LIN {X 0,Y 233.584,Z 324.878,A -85,B 0,C 180,E1 -20817.651,E2 -20817.651} C_VEL
LIN {X 0,Y 230.113,Z 315.653,A -85,B 0,C 180,E1 -20819.516,E2 -20819.516} C_VEL
LIN {X 0,Y 226.325,Z 305.069,A -85,B 0,C 180,E1 -20821.384,E2 -20821.384} C_VEL
LIN {X 0,Y 221.321,Z 294.088,A -85,B 0,C 180,E1 -20823.248,E2 -20823.248} C_VEL
LIN {X 0,Y 216.634,Z 285.381,A -85,B 0,C 180,E1 -20824.719,E2 -20824.719} C_VEL
LIN {X 0,Y 215.299,Z 283.034,A -85,B 0,C 180,E1 -20825.102,E2 -20825.102} C_VEL
LIN {X 0,Y 213.881,Z 280.332,A -85,B 0,C 180,E1 -20825.505,E2 -20825.505} C_VEL
LIN {X 0,Y 213.692,Z 279.368,A -85,B 0,C 180,E1 -20825.598,E2 -20825.598} C_VEL
LIN {X 0,Y 213.741,Z 279.36,A -85,B 0,C 180,E1 -20828.662,E2 -20828.662} C_VEL
LIN {X 0,Y 213.757,Z 279.358,A -85,B 0,C 180,E1 -20831.114,E2 -20831.114} C_VEL
LIN {X 0,Y 213.799,Z 279.355,A -85,B 0,C 180,E1 -20833.702,E2 -20833.702} C_VEL
LIN {X 0,Y 213.776,Z 279.356,A -85,B 0,C 180,E1 -20836.358,E2 -20836.358} C_VEL
LIN {X 0,Y 213.763,Z 279.358,A -85,B 0,C 180,E1 -20839.128,E2 -20839.128} C_VEL
LIN {X 0,Y 213.723,Z 279.362,A -85,B 0,C 180,E1 -20843.724,E2 -20843.724} C_VEL
LIN {X 0,Y 213.769,Z 279.357,A -85,B 0,C 180,E1 -20848.735,E2 -20848.735} C_VEL
LIN {X 0,Y 213.802,Z 279.353,A -85,B 0,C 180,E1 -20852.614,E2 -20852.614} C_VEL
LIN {X 0,Y 213.797,Z 279.354,A -85,B 0,C 180,E1 -20856.985,E2 -20856.985} C_VEL
LIN {X 0,Y 213.876,Z 279.345,A -85,B 0,C 180,E1 -20862.811,E2 -20862.811} C_VEL
LIN {X 0,Y 213.921,Z 279.337,A -85,B 0,C 180,E1 -20866.717,E2 -20866.717} C_VEL
LIN {X 0,Y 214.127,Z 279.307,A -85,B 0,C 180,E1 -20870.566,E2 -20870.566} C_VEL
LIN {X 0,Y 214.076,Z 279.315,A -85,B 0,C 180,E1 -20874.359,E2 -20874.359} C_VEL
LIN {X 0,Y 214.402,Z 279.25,A -85,B 0,C 180,E1 -20878.133,E2 -20878.133} C_VEL
LIN {X 0,Y 214.507,Z 279.25,A -85,B 0,C 180,E1 -20880.011,E2 -20880.011} C_VEL
LIN {X 0,Y 214.401,Z 279.275,A -85,B 0,C 180,E1 -20881.889,E2 -20881.889} C_VEL
LIN {X 0,Y 214.183,Z 279.306,A -85,B 0,C 180,E1 -20887.553,E2 -20887.553} C_VEL
LIN {X 0,Y 213.985,Z 279.33,A -85,B 0,C 180,E1 -20891.376,E2 -20891.376} C_VEL
LIN {X 0,Y 213.876,Z 279.344,A -85,B 0,C 180,E1 -20895.251,E2 -20895.251} C_VEL
LIN {X 0,Y 213.798,Z 279.354,A -85,B 0,C 180,E1 -20899.202,E2 -20899.202} C_VEL
LIN {X 0,Y 213.774,Z 279.359,A -85,B 0,C 180,E1 -20903.246,E2 -20903.246} C_VEL
LIN {X 0,Y 213.84,Z 279.719,A -85,B 0,C 180,E1 -20907.405,E2 -20907.405} C_VEL
LIN {X 0,Y 214.016,Z 281.418,A -85,B 0,C 180,E1 -20911.707,E2 -20911.707} C_VEL
LIN {X 0,Y 214.301,Z 283.414,A -85,B 0,C 180,E1 -20916.19,E2 -20916.19} C_VEL
LIN {X 0,Y 214.677,Z 285.89,A -85,B 0,C 180,E1 -20921.153,E2 -20921.153} C_VEL
LIN {X 0,Y 214.856,Z 287.42,A -85,B 0,C 180,E1 -20923.977,E2 -20923.977} C_VEL
LIN {X 0,Y 214.874,Z 288.962,A -85,B 0,C 180,E1 -20926.619,E2 -20926.619} C_VEL
LIN {X 0,Y 214.706,Z 290.501,A -85,B 0,C 180,E1 -20929.107,E2 -20929.107} C_VEL
LIN {X 0,Y 214.243,Z 292.34,A -85,B 0,C 180,E1 -20931.946,E2 -20931.946} C_VEL
LIN {X 0,Y 213.723,Z 294.297,A -85,B 0,C 180,E1 -20934.668,E2 -20934.668} C_VEL
LIN {X 0,Y 214.726,Z 297.663,A -85,B 0,C 180,E1 -20935.037,E2 -20935.037} C_VEL
LIN {X 0,Y 218.182,Z 307.912,A -85,B 0,C 180,E1 -20936.445,E2 -20936.445} C_VEL
LIN {X 0,Y 221.383,Z 321.092,A -85,B 0,C 180,E1 -20938.39,E2 -20938.39} C_VEL
LIN {X 0,Y 222.985,Z 331.539,A -85,B 0,C 180,E1 -20940.079,E2 -20940.079} C_VEL
LIN {X 0,Y 223.807,Z 339.866,A -85,B 0,C 180,E1 -20941.568,E2 -20941.568} C_VEL
LIN {X 0,Y 223.951,Z 349.305,A -85,B 0,C 180,E1 -20943.44,E2 -20943.44} C_VEL
LIN {X 0,Y 223.681,Z 353.86,A -85,B 0,C 180,E1 -20944.405,E2 -20944.405} C_VEL
LIN {X 0,Y 220.756,Z 364.316,A -85,B 0,C 180,E1 -20946.817,E2 -20946.817} C_VEL
LIN {X 0,Y 218.8,Z 371.499,A -85,B 0,C 180,E1 -20948.896,E2 -20948.896} C_VEL
LIN {X 0,Y 216.843,Z 377.815,A -85,B 0,C 180,E1 -20951.089,E2 -20951.089} C_VEL
LIN {X 0,Y 215.402,Z 382.705,A -85,B 0,C 180,E1 -20953.12,E2 -20953.12} C_VEL
LIN {X 0,Y 213.879,Z 385.575,A -85,B 0,C 180,E1 -20954.456,E2 -20954.456} C_VEL
LIN {X 0,Y 209.871,Z 389.592,A -85,B 0,C 180,E1 -20956.645,E2 -20956.645} C_VEL
LIN {X 0,Y 206.107,Z 393.022,A -85,B 0,C 180,E1 -20958.99,E2 -20958.99} C_VEL
LIN {X 0,Y 204.997,Z 394.677,A -85,B 0,C 180,E1 -20960.54,E2 -20960.54} C_VEL
LIN {X 0,Y 204.442,Z 397.502,A -85,B 0,C 180,E1 -20964.081,E2 -20964.081} C_VEL
LIN {X 0,Y 204.364,Z 398.567,A -85,B 0,C 180,E1 -20966.056,E2 -20966.056} C_VEL
LIN {X 0,Y 204.351,Z 399.161,A -85,B 0,C 180,E1 -20968.029,E2 -20968.029} C_VEL
LIN {X 0,Y 204.44,Z 399.319,A -85,B 0,C 180,E1 -20970,E2 -20970} C_VEL
LIN {X 0,Y 204.351,Z 399.161,A -85,B 0,C 180,E1 -20971.971,E2 -20971.971} C_VEL
LIN {X 0,Y 204.374,Z 398.506,A -85,B 0,C 180,E1 -20974.143,E2 -20974.143} C_VEL
LIN {X 0,Y 204.692,Z 396.109,A -85,B 0,C 180,E1 -20977.894,E2 -20977.894} C_VEL
LIN {X 0,Y 205.364,Z 393.153,A -85,B 0,C 180,E1 -20980.849,E2 -20980.849} C_VEL
LIN {X 0,Y 206.41,Z 389.156,A -85,B 0,C 180,E1 -20983.788,E2 -20983.788} C_VEL
LIN {X 0,Y 208.054,Z 384.024,A -85,B 0,C 180,E1 -20986.686,E2 -20986.686} C_VEL
LIN {X 0,Y 209.72,Z 378.758,A -85,B 0,C 180,E1 -20989.07,E2 -20989.07} C_VEL
LIN {X 0,Y 211.801,Z 372.441,A -85,B 0,C 180,E1 -20991.407,E2 -20991.407} C_VEL
LIN {X 0,Y 213.504,Z 366.484,A -85,B 0,C 180,E1 -20993.266,E2 -20993.266} C_VEL
LIN {X 0,Y 215.522,Z 359.556,A -85,B 0,C 180,E1 -20995.082,E2 -20995.082} C_VEL
LIN {X 0,Y 217.202,Z 353.645,A -85,B 0,C 180,E1 -20996.417,E2 -20996.417} C_VEL
LIN {X 0,Y 217.35,Z 343.883,A -85,B 0,C 180,E1 -20998.535,E2 -20998.535} C_VEL
LIN {X 0,Y 216.713,Z 334.568,A -85,B 0,C 180,E1 -21000.347,E2 -21000.347} C_VEL
LIN {X 0,Y 215.482,Z 325.215,A -85,B 0,C 180,E1 -21001.991,E2 -21001.991} C_VEL
LIN {X 0,Y 213.725,Z 316.4,A -85,B 0,C 180,E1 -21003.43,E2 -21003.43} C_VEL
LIN {X 0,Y 210.705,Z 305.251,A -85,B 0,C 180,E1 -21005.113,E2 -21005.113} C_VEL
LIN {X 0,Y 207.594,Z 296.756,A -85,B 0,C 180,E1 -21006.388,E2 -21006.388} C_VEL
LIN {X 0,Y 206.912,Z 293.968,A -85,B 0,C 180,E1 -21006.722,E2 -21006.722} C_VEL
LIN {X 0,Y 207.477,Z 291.775,A -85,B 0,C 180,E1 -21010.06,E2 -21010.06} C_VEL
LIN {X 0,Y 207.716,Z 290.247,A -85,B 0,C 180,E1 -21012.585,E2 -21012.585} C_VEL
LIN {X 0,Y 207.776,Z 288.728,A -85,B 0,C 180,E1 -21015.26,E2 -21015.26} C_VEL
LIN {X 0,Y 207.669,Z 287.189,A -85,B 0,C 180,E1 -21018.118,E2 -21018.118} C_VEL
LIN {X 0,Y 207.355,Z 285.063,A -85,B 0,C 180,E1 -21022.393,E2 -21022.393} C_VEL
LIN {X 0,Y 207.219,Z 283.979,A -85,B 0,C 180,E1 -21024.779,E2 -21024.779} C_VEL
LIN {X 0,Y 206.936,Z 282.067,A -85,B 0,C 180,E1 -21029.363,E2 -21029.363} C_VEL
LIN {X 0,Y 206.712,Z 280.437,A -85,B 0,C 180,E1 -21033.758,E2 -21033.758} C_VEL
LIN {X 0,Y 206.716,Z 280.242,A -85,B 0,C 180,E1 -21038.028,E2 -21038.028} C_VEL
LIN {X 0,Y 206.811,Z 280.226,A -85,B 0,C 180,E1 -21042.18,E2 -21042.18} C_VEL
LIN {X 0,Y 206.858,Z 280.219,A -85,B 0,C 180,E1 -21046.231,E2 -21046.231} C_VEL
LIN {X 0,Y 207.08,Z 280.192,A -85,B 0,C 180,E1 -21050.219,E2 -21050.219} C_VEL
LIN {X 0,Y 207.036,Z 280.196,A -85,B 0,C 180,E1 -21054.144,E2 -21054.144} C_VEL
LIN {X 0,Y 207.341,Z 280.155,A -85,B 0,C 180,E1 -21058.046,E2 -21058.046} C_VEL
LIN {X 0,Y 207.475,Z 280.125,A -85,B 0,C 180,E1 -21059.989,E2 -21059.989} C_VEL
LIN {X 0,Y 207.342,Z 280.128,A -85,B 0,C 180,E1 -21061.931,E2 -21061.931} C_VEL
LIN {X 0,Y 207.123,Z 280.184,A -85,B 0,C 180,E1 -21067.789,E2 -21067.789} C_VEL
LIN {X 0,Y 206.904,Z 280.213,A -85,B 0,C 180,E1 -21071.747,E2 -21071.747} C_VEL
LIN {X 0,Y 206.814,Z 280.22,A -85,B 0,C 180,E1 -21075.762,E2 -21075.762} C_VEL
LIN {X 0,Y 206.714,Z 280.228,A -85,B 0,C 180,E1 -21079.863,E2 -21079.863} C_VEL
LIN {X 0,Y 206.725,Z 280.231,A -85,B 0,C 180,E1 -21084.063,E2 -21084.063} C_VEL
LIN {X 0,Y 206.719,Z 280.235,A -85,B 0,C 180,E1 -21088.408,E2 -21088.408} C_VEL
LIN {X 0,Y 206.68,Z 280.239,A -85,B 0,C 180,E1 -21092.945,E2 -21092.945} C_VEL
LIN {X 0,Y 206.693,Z 280.238,A -85,B 0,C 180,E1 -21097.72,E2 -21097.72} C_VEL
LIN {X 0,Y 206.691,Z 280.238,A -85,B 0,C 180,E1 -21101.579,E2 -21101.579} C_VEL
LIN {X 0,Y 206.709,Z 280.235,A -85,B 0,C 180,E1 -21105.541,E2 -21105.541} C_VEL
LIN {X 0,Y 206.686,Z 280.238,A -85,B 0,C 180,E1 -21109.756,E2 -21109.756} C_VEL
LIN {X 0,Y 206.675,Z 280.3,A -85,B 0,C 180,E1 -21113.049,E2 -21113.049} C_VEL
LIN {X 0,Y 207.645,Z 283.045,A -85,B 0,C 180,E1 -21113.409,E2 -21113.409} C_VEL
LIN {X 0,Y 209.134,Z 285.264,A -85,B 0,C 180,E1 -21113.839,E2 -21113.839} C_VEL
LIN {X 0,Y 214.621,Z 295.422,A -85,B 0,C 180,E1 -21115.662,E2 -21115.662} C_VEL
LIN {X 0,Y 220.071,Z 307.47,A -85,B 0,C 180,E1 -21117.86,E2 -21117.86} C_VEL
LIN {X 0,Y 223.998,Z 318.702,A -85,B 0,C 180,E1 -21120.011,E2 -21120.011} C_VEL
LIN {X 0,Y 226.852,Z 326.94,A -85,B 0,C 180,E1 -21121.772,E2 -21121.772} C_VEL
LIN {X 0,Y 230.624,Z 335.068,A -85,B 0,C 180,E1 -21123.819,E2 -21123.819} C_VEL
LIN {X 0,Y 235.907,Z 343.688,A -85,B 0,C 180,E1 -21126.327,E2 -21126.327} C_VEL
LIN {X 0,Y 242.775,Z 352.2,A -85,B 0,C 180,E1 -21129.194,E2 -21129.194} C_VEL
LIN {X 0,Y 250.909,Z 359.994,A -85,B 0,C 180,E1 -21132.199,E2 -21132.199} C_VEL
LIN {X 0,Y 258.449,Z 366.061,A -85,B 0,C 180,E1 -21134.823,E2 -21134.823} C_VEL
LIN {X 0,Y 267.552,Z 372.22,A -85,B 0,C 180,E1 -21137.87,E2 -21137.87} C_VEL
LIN {X 0,Y 274.83,Z 376.627,A -85,B 0,C 180,E1 -21140.432,E2 -21140.432} C_VEL
LIN {X 0,Y 280.808,Z 379.995,A -85,B 0,C 180,E1 -21142.811,E2 -21142.811} C_VEL
LIN {X 0,Y 283.757,Z 381.703,A -85,B 0,C 180,E1 -21144.314,E2 -21144.314} C_VEL
LIN {X 0,Y 285.917,Z 383.016,A -85,B 0,C 180,E1 -21145.771,E2 -21145.771} C_VEL
LIN {X 0,Y 288.366,Z 384.106,A -85,B 0,C 180,E1 -21147.49,E2 -21147.49} C_VEL
LIN {X 0,Y 289.55,Z 384.495,A -85,B 0,C 180,E1 -21148.609,E2 -21148.609} C_VEL
LIN {X 0,Y 290.56,Z 384.663,A -85,B 0,C 180,E1 -21150,E2 -21150} C_VEL
LIN {X 0,Y 289.541,Z 384.496,A -85,B 0,C 180,E1 -21151.391,E2 -21151.391} C_VEL
LIN {X 0,Y 287.923,Z 383.952,A -85,B 0,C 180,E1 -21152.798,E2 -21152.798} C_VEL
LIN {X 0,Y 285.915,Z 383.015,A -85,B 0,C 180,E1 -21154.229,E2 -21154.229} C_VEL
LIN {X 0,Y 282.759,Z 381.067,A -85,B 0,C 180,E1 -21156.282,E2 -21156.282} C_VEL
LIN {X 0,Y 280.804,Z 379.995,A -85,B 0,C 180,E1 -21157.189,E2 -21157.189} C_VEL
LIN {X 0,Y 274.84,Z 376.626,A -85,B 0,C 180,E1 -21159.568,E2 -21159.568} C_VEL
LIN {X 0,Y 267.586,Z 372.219,A -85,B 0,C 180,E1 -21162.129,E2 -21162.129} C_VEL
LIN {X 0,Y 258.457,Z 366.04,A -85,B 0,C 180,E1 -21165.184,E2 -21165.184} C_VEL
LIN {X 0,Y 250.411,Z 359.547,A -85,B 0,C 180,E1 -21167.982,E2 -21167.982} C_VEL
LIN {X 0,Y 242.793,Z 352.219,A -85,B 0,C 180,E1 -21170.799,E2 -21170.799} C_VEL
LIN {X 0,Y 235.891,Z 343.734,A -85,B 0,C 180,E1 -21173.664,E2 -21173.664} C_VEL
LIN {X 0,Y 230.636,Z 335.053,A -85,B 0,C 180,E1 -21176.183,E2 -21176.183} C_VEL
LIN {X 0,Y 226.877,Z 326.928,A -85,B 0,C 180,E1 -21178.226,E2 -21178.226} C_VEL
LIN {X 0,Y 223.241,Z 316.351,A -85,B 0,C 180,E1 -21180.456,E2 -21180.456} C_VEL
LIN {X 0,Y 219.366,Z 305.777,A -85,B 0,C 180,E1 -21182.448,E2 -21182.448} C_VEL
LIN {X 0,Y 214.168,Z 294.426,A -85,B 0,C 180,E1 -21184.504,E2 -21184.504} C_VEL
LIN {X 0,Y 208.413,Z 284.067,A -85,B 0,C 180,E1 -21186.397,E2 -21186.397} C_VEL
LIN {X 0,Y 206.985,Z 281.663,A -85,B 0,C 180,E1 -21186.823,E2 -21186.823} C_VEL
LIN {X 0,Y 206.658,Z 280.243,A -85,B 0,C 180,E1 -21187.019,E2 -21187.019} C_VEL
LIN {X 0,Y 206.686,Z 280.238,A -85,B 0,C 180,E1 -21190.244,E2 -21190.244} C_VEL
LIN {X 0,Y 206.709,Z 280.235,A -85,B 0,C 180,E1 -21194.459,E2 -21194.459} C_VEL
LIN {X 0,Y 206.691,Z 280.238,A -85,B 0,C 180,E1 -21198.421,E2 -21198.421} C_VEL
LIN {X 0,Y 206.693,Z 280.238,A -85,B 0,C 180,E1 -21202.28,E2 -21202.28} C_VEL
LIN {X 0,Y 206.68,Z 280.239,A -85,B 0,C 180,E1 -21207.055,E2 -21207.055} C_VEL
LIN {X 0,Y 206.742,Z 280.232,A -85,B 0,C 180,E1 -21212.108,E2 -21212.108} C_VEL
LIN {X 0,Y 206.732,Z 280.232,A -85,B 0,C 180,E1 -21216.616,E2 -21216.616} C_VEL
LIN {X 0,Y 206.808,Z 280.223,A -85,B 0,C 180,E1 -21222.204,E2 -21222.204} C_VEL
LIN {X 0,Y 206.861,Z 280.214,A -85,B 0,C 180,E1 -21226.255,E2 -21226.255} C_VEL
LIN {X 0,Y 207.07,Z 280.185,A -85,B 0,C 180,E1 -21230.242,E2 -21230.242} C_VEL
LIN {X 0,Y 207.038,Z 280.193,A -85,B 0,C 180,E1 -21234.167,E2 -21234.167} C_VEL
LIN {X 0,Y 207.342,Z 280.128,A -85,B 0,C 180,E1 -21238.069,E2 -21238.069} C_VEL
LIN {X 0,Y 207.475,Z 280.125,A -85,B 0,C 180,E1 -21240.011,E2 -21240.011} C_VEL
LIN {X 0,Y 207.341,Z 280.155,A -85,B 0,C 180,E1 -21241.954,E2 -21241.954} C_VEL
LIN {X 0,Y 207.127,Z 280.186,A -85,B 0,C 180,E1 -21247.811,E2 -21247.811} C_VEL
LIN {X 0,Y 206.906,Z 280.214,A -85,B 0,C 180,E1 -21251.77,E2 -21251.77} C_VEL
LIN {X 0,Y 206.81,Z 280.226,A -85,B 0,C 180,E1 -21255.786,E2 -21255.786} C_VEL
LIN {X 0,Y 206.719,Z 280.237,A -85,B 0,C 180,E1 -21259.886,E2 -21259.886} C_VEL
LIN {X 0,Y 206.702,Z 280.238,A -85,B 0,C 180,E1 -21264.091,E2 -21264.091} C_VEL
LIN {X 0,Y 206.718,Z 280.43,A -85,B 0,C 180,E1 -21266.241,E2 -21266.241} C_VEL
LIN {X 0,Y 206.938,Z 282.065,A -85,B 0,C 180,E1 -21270.637,E2 -21270.637} C_VEL
LIN {X 0,Y 207.246,Z 284.124,A -85,B 0,C 180,E1 -21275.525,E2 -21275.525} C_VEL
LIN {X 0,Y 207.534,Z 286.286,A -85,B 0,C 180,E1 -21280.059,E2 -21280.059} C_VEL
LIN {X 0,Y 207.707,Z 287.575,A -85,B 0,C 180,E1 -21282.6,E2 -21282.6} C_VEL
LIN {X 0,Y 207.804,Z 289.026,A -85,B 0,C 180,E1 -21285.266,E2 -21285.266} C_VEL
LIN {X 0,Y 207.678,Z 290.699,A -85,B 0,C 180,E1 -21288.129,E2 -21288.129} C_VEL
LIN {X 0,Y 207.281,Z 292.617,A -85,B 0,C 180,E1 -21291.259,E2 -21291.259} C_VEL
LIN {X 0,Y 206.883,Z 293.954,A -85,B 0,C 180,E1 -21293.284,E2 -21293.284} C_VEL
LIN {X 0,Y 207.798,Z 297.248,A -85,B 0,C 180,E1 -21293.681,E2 -21293.681} C_VEL
LIN {X 0,Y 211.704,Z 308.489,A -85,B 0,C 180,E1 -21295.347,E2 -21295.347} C_VEL
LIN {X 0,Y 214.523,Z 319.927,A -85,B 0,C 180,E1 -21297.128,E2 -21297.128} C_VEL
LIN {X 0,Y 216.188,Z 329.971,A -85,B 0,C 180,E1 -21298.817,E2 -21298.817} C_VEL
LIN {X 0,Y 217.112,Z 339.358,A -85,B 0,C 180,E1 -21300.552,E2 -21300.552} C_VEL
LIN {X 0,Y 217.361,Z 348.332,A -85,B 0,C 180,E1 -21302.396,E2 -21302.396} C_VEL
LIN {X 0,Y 216.99,Z 354.737,A -85,B 0,C 180,E1 -21303.814,E2 -21303.814} C_VEL
LIN {X 0,Y 214.49,Z 363.229,A -85,B 0,C 180,E1 -21305.822,E2 -21305.822} C_VEL
LIN {X 0,Y 212.24,Z 370.767,A -85,B 0,C 180,E1 -21308.02,E2 -21308.02} C_VEL
LIN {X 0,Y 210.12,Z 377.603,A -85,B 0,C 180,E1 -21310.46,E2 -21310.46} C_VEL
LIN {X 0,Y 208.474,Z 382.847,A -85,B 0,C 180,E1 -21312.729,E2 -21312.729} C_VEL
LIN {X 0,Y 206.896,Z 387.601,A -85,B 0,C 180,E1 -21315.241,E2 -21315.241} C_VEL
LIN {X 0,Y 205.669,Z 391.933,A -85,B 0,C 180,E1 -21318.169,E2 -21318.169} C_VEL
LIN {X 0,Y 204.997,Z 394.677,A -85,B 0,C 180,E1 -21320.54,E2 -21320.54} C_VEL
LIN {X 0,Y 203.994,Z 396.162,A -85,B 0,C 180,E1 -21322.128,E2 -21322.128} C_VEL
LIN {X 0,Y 200.819,Z 397.852,A -85,B 0,C 180,E1 -21324.746,E2 -21324.746} C_VEL
LIN {X 0,Y 198.332,Z 398.675,A -85,B 0,C 180,E1 -21326.911,E2 -21326.911} C_VEL
LIN {X 0,Y 197.286,Z 399.105,A -85,B 0,C 180,E1 -21328.895,E2 -21328.895} C_VEL
LIN {X 0,Y 197.279,Z 399.044,A -85,B 0,C 180,E1 -21329.183,E2 -21329.183} C_VEL
LIN {X 0,Y 197.26,Z 398.949,A -85,B 0,C 180,E1 -21332.042,E2 -21332.042} C_VEL
LIN {X 0,Y 197.277,Z 398.356,A -85,B 0,C 180,E1 -21334.086,E2 -21334.086} C_VEL
LIN {X 0,Y 197.638,Z 395.897,A -85,B 0,C 180,E1 -21338.177,E2 -21338.177} C_VEL
LIN {X 0,Y 198.353,Z 392.94,A -85,B 0,C 180,E1 -21341.237,E2 -21341.237} C_VEL
LIN {X 0,Y 199.481,Z 388.944,A -85,B 0,C 180,E1 -21344.277,E2 -21344.277} C_VEL
LIN {X 0,Y 201.235,Z 383.812,A -85,B 0,C 180,E1 -21347.269,E2 -21347.269} C_VEL
LIN {X 0,Y 202.995,Z 378.546,A -85,B 0,C 180,E1 -21349.728,E2 -21349.728} C_VEL
LIN {X 0,Y 205.164,Z 372.229,A -85,B 0,C 180,E1 -21352.136,E2 -21352.136} C_VEL
LIN {X 0,Y 206.962,Z 366.272,A -85,B 0,C 180,E1 -21354.047,E2 -21354.047} C_VEL
LIN {X 0,Y 209.084,Z 359.344,A -85,B 0,C 180,E1 -21355.91,E2 -21355.91} C_VEL
LIN {X 0,Y 210.541,Z 354.522,A -85,B 0,C 180,E1 -21357.052,E2 -21357.052} C_VEL
LIN {X 0,Y 210.757,Z 343.659,A -85,B 0,C 180,E1 -21359.514,E2 -21359.514} C_VEL
LIN {X 0,Y 210.214,Z 335.056,A -85,B 0,C 180,E1 -21361.268,E2 -21361.268} C_VEL
LIN {X 0,Y 208.933,Z 325.243,A -85,B 0,C 180,E1 -21363.083,E2 -21363.083} C_VEL
LIN {X 0,Y 206.822,Z 315.118,A -85,B 0,C 180,E1 -21364.82,E2 -21364.82} C_VEL
LIN {X 0,Y 203.979,Z 305.168,A -85,B 0,C 180,E1 -21366.438,E2 -21366.438} C_VEL
LIN {X 0,Y 201.116,Z 297.224,A -85,B 0,C 180,E1 -21367.718,E2 -21367.718} C_VEL
LIN {X 0,Y 200.137,Z 294.243,A -85,B 0,C 180,E1 -21368.111,E2 -21368.111} C_VEL
LIN {X 0,Y 200.129,Z 293.719,A -85,B 0,C 180,E1 -21368.233,E2 -21368.233} C_VEL
LIN {X 0,Y 200.664,Z 291.036,A -85,B 0,C 180,E1 -21372.637,E2 -21372.637} C_VEL
LIN {X 0,Y 200.705,Z 289.436,A -85,B 0,C 180,E1 -21375.533,E2 -21375.533} C_VEL
LIN {X 0,Y 200.626,Z 288.029,A -85,B 0,C 180,E1 -21378.261,E2 -21378.261} C_VEL
LIN {X 0,Y 200.237,Z 285.623,A -85,B 0,C 180,E1 -21383.356,E2 -21383.356} C_VEL
LIN {X 0,Y 199.97,Z 283.597,A -85,B 0,C 180,E1 -21388.173,E2 -21388.173} C_VEL
LIN {X 0,Y 199.738,Z 281.898,A -85,B 0,C 180,E1 -21392.768,E2 -21392.768} C_VEL
LIN {X 0,Y 199.637,Z 281.153,A -85,B 0,C 180,E1 -21395,E2 -21395} C_VEL
LIN {X 0,Y 199.65,Z 281.12,A -85,B 0,C 180,E1 -21399.378,E2 -21399.378} C_VEL
LIN {X 0,Y 199.749,Z 281.104,A -85,B 0,C 180,E1 -21403.641,E2 -21403.641} C_VEL
LIN {X 0,Y 200.027,Z 281.07,A -85,B 0,C 180,E1 -21409.871,E2 -21409.871} C_VEL
LIN {X 0,Y 200,Z 281.073,A -85,B 0,C 180,E1 -21413.937,E2 -21413.937} C_VEL
LIN {X 0,Y 200.283,Z 281.034,A -85,B 0,C 180,E1 -21417.977,E2 -21417.977} C_VEL
LIN {X 0,Y 200.442,Z 281,A -85,B 0,C 180,E1 -21419.988,E2 -21419.988} C_VEL
LIN {X 0,Y 199.991,Z 281.055,A -85,B 0,C 180,E1 -21424.018,E2 -21424.018} C_VEL
LIN {X 0,Y 200.07,Z 281.061,A -85,B 0,C 180,E1 -21428.065,E2 -21428.065} C_VEL
LIN {X 0,Y 199.853,Z 281.09,A -85,B 0,C 180,E1 -21432.168,E2 -21432.168} C_VEL
LIN {X 0,Y 199.75,Z 281.101,A -85,B 0,C 180,E1 -21436.335,E2 -21436.335} C_VEL
LIN {X 0,Y 199.644,Z 281.109,A -85,B 0,C 180,E1 -21440.597,E2 -21440.597} C_VEL
LIN {X 0,Y 199.642,Z 281.11,A -85,B 0,C 180,E1 -21444.974,E2 -21444.974} C_VEL
LIN {X 0,Y 199.649,Z 281.116,A -85,B 0,C 180,E1 -21449.511,E2 -21449.511} C_VEL
LIN {X 0,Y 199.636,Z 281.118,A -85,B 0,C 180,E1 -21452.341,E2 -21452.341} C_VEL
LIN {X 0,Y 199.622,Z 281.12,A -85,B 0,C 180,E1 -21456.746,E2 -21456.746} C_VEL
LIN {X 0,Y 199.646,Z 281.116,A -85,B 0,C 180,E1 -21459.301,E2 -21459.301} C_VEL
LIN {X 0,Y 199.629,Z 281.118,A -85,B 0,C 180,E1 -21462.328,E2 -21462.328} C_VEL
LIN {X 0,Y 199.657,Z 281.113,A -85,B 0,C 180,E1 -21465.252,E2 -21465.252} C_VEL
LIN {X 0,Y 199.629,Z 281.118,A -85,B 0,C 180,E1 -21468.019,E2 -21468.019} C_VEL
LIN {X 0,Y 199.677,Z 281.113,A -85,B 0,C 180,E1 -21471.529,E2 -21471.529} C_VEL
LIN {X 0,Y 200.769,Z 284.157,A -85,B 0,C 180,E1 -21471.989,E2 -21471.989} C_VEL
LIN {X 0,Y 202.251,Z 286.351,A -85,B 0,C 180,E1 -21472.45,E2 -21472.45} C_VEL
LIN {X 0,Y 208.099,Z 296.985,A -85,B 0,C 180,E1 -21474.541,E2 -21474.541} C_VEL
LIN {X 0,Y 213.126,Z 308.109,A -85,B 0,C 180,E1 -21476.73,E2 -21476.73} C_VEL
LIN {X 0,Y 216.72,Z 318.012,A -85,B 0,C 180,E1 -21478.745,E2 -21478.745} C_VEL
LIN {X 0,Y 220.11,Z 328.756,A -85,B 0,C 180,E1 -21481.131,E2 -21481.131} C_VEL
LIN {X 0,Y 223.354,Z 336.507,A -85,B 0,C 180,E1 -21483.151,E2 -21483.151} C_VEL
LIN {X 0,Y 228.441,Z 345.263,A -85,B 0,C 180,E1 -21485.839,E2 -21485.839} C_VEL
LIN {X 0,Y 234.148,Z 352.752,A -85,B 0,C 180,E1 -21488.472,E2 -21488.472} C_VEL
LIN {X 0,Y 241.109,Z 359.831,A -85,B 0,C 180,E1 -21491.299,E2 -21491.299} C_VEL
LIN {X 0,Y 248.491,Z 365.896,A -85,B 0,C 180,E1 -21494.027,E2 -21494.027} C_VEL
LIN {X 0,Y 255.952,Z 371.045,A -85,B 0,C 180,E1 -21496.636,E2 -21496.636} C_VEL
LIN {X 0,Y 264.379,Z 376.003,A -85,B 0,C 180,E1 -21499.532,E2 -21499.532} C_VEL
LIN {X 0,Y 269.921,Z 378.947,A -85,B 0,C 180,E1 -21501.573,E2 -21501.573} C_VEL
LIN {X 0,Y 275.574,Z 381.733,A -85,B 0,C 180,E1 -21503.941,E2 -21503.941} C_VEL
LIN {X 0,Y 278.37,Z 383.239,A -85,B 0,C 180,E1 -21505.656,E2 -21505.656} C_VEL
LIN {X 0,Y 281.29,Z 384.422,A -85,B 0,C 180,E1 -21507.693,E2 -21507.693} C_VEL
LIN {X 0,Y 282.26,Z 384.711,A -85,B 0,C 180,E1 -21508.573,E2 -21508.573} C_VEL
LIN {X 0,Y 283.391,Z 384.873,A -85,B 0,C 180,E1 -21510,E2 -21510} C_VEL
LIN {X 0,Y 282.247,Z 384.712,A -85,B 0,C 180,E1 -21511.427,E2 -21511.427} C_VEL
LIN {X 0,Y 280.451,Z 384.176,A -85,B 0,C 180,E1 -21512.873,E2 -21512.873} C_VEL
LIN {X 0,Y 278.368,Z 383.239,A -85,B 0,C 180,E1 -21514.344,E2 -21514.344} C_VEL
LIN {X 0,Y 275.574,Z 381.733,A -85,B 0,C 180,E1 -21516.059,E2 -21516.059} C_VEL
LIN {X 0,Y 269.921,Z 378.947,A -85,B 0,C 180,E1 -21518.426,E2 -21518.426} C_VEL
LIN {X 0,Y 263.546,Z 375.53,A -85,B 0,C 180,E1 -21520.758,E2 -21520.758} C_VEL
LIN {X 0,Y 255.958,Z 371.038,A -85,B 0,C 180,E1 -21523.367,E2 -21523.367} C_VEL
LIN {X 0,Y 246.924,Z 364.712,A -85,B 0,C 180,E1 -21526.536,E2 -21526.536} C_VEL
LIN {X 0,Y 237.567,Z 356.446,A -85,B 0,C 180,E1 -21530.11,E2 -21530.11} C_VEL
LIN {X 0,Y 230.868,Z 348.775,A -85,B 0,C 180,E1 -21532.984,E2 -21532.984} C_VEL
LIN {X 0,Y 225.798,Z 340.98,A -85,B 0,C 180,E1 -21535.526,E2 -21535.526} C_VEL
LIN {X 0,Y 222.082,Z 333.564,A -85,B 0,C 180,E1 -21537.644,E2 -21537.644} C_VEL
LIN {X 0,Y 218.713,Z 324.59,A -85,B 0,C 180,E1 -21539.847,E2 -21539.847} C_VEL
LIN {X 0,Y 215.45,Z 314.226,A -85,B 0,C 180,E1 -21542.018,E2 -21542.018} C_VEL
LIN {X 0,Y 211.674,Z 304.797,A -85,B 0,C 180,E1 -21543.921,E2 -21543.921} C_VEL
LIN {X 0,Y 207.125,Z 295.195,A -85,B 0,C 180,E1 -21545.808,E2 -21545.808} C_VEL
LIN {X 0,Y 203.074,Z 287.944,A -85,B 0,C 180,E1 -21547.275,E2 -21547.275} C_VEL
LIN {X 0,Y 201.459,Z 285.033,A -85,B 0,C 180,E1 -21547.824,E2 -21547.824} C_VEL
LIN {X 0,Y 199.989,Z 282.483,A -85,B 0,C 180,E1 -21548.309,E2 -21548.309} C_VEL
LIN {X 0,Y 199.682,Z 281.112,A -85,B 0,C 180,E1 -21548.535,E2 -21548.535} C_VEL
LIN {X 0,Y 199.625,Z 281.117,A -85,B 0,C 180,E1 -21552.347,E2 -21552.347} C_VEL
LIN {X 0,Y 199.657,Z 281.114,A -85,B 0,C 180,E1 -21555.271,E2 -21555.271} C_VEL
LIN {X 0,Y 199.633,Z 281.119,A -85,B 0,C 180,E1 -21558.038,E2 -21558.038} C_VEL
LIN {X 0,Y 199.648,Z 281.116,A -85,B 0,C 180,E1 -21560.753,E2 -21560.753} C_VEL
LIN {X 0,Y 199.606,Z 281.121,A -85,B 0,C 180,E1 -21565.729,E2 -21565.729} C_VEL
LIN {X 0,Y 199.676,Z 281.112,A -85,B 0,C 180,E1 -21568.149,E2 -21568.149} C_VEL
LIN {X 0,Y 199.663,Z 281.115,A -85,B 0,C 180,E1 -21572.783,E2 -21572.783} C_VEL
LIN {X 0,Y 199.692,Z 281.112,A -85,B 0,C 180,E1 -21577.238,E2 -21577.238} C_VEL
LIN {X 0,Y 199.733,Z 281.104,A -85,B 0,C 180,E1 -21581.811,E2 -21581.811} C_VEL
LIN {X 0,Y 199.799,Z 281.092,A -85,B 0,C 180,E1 -21585.759,E2 -21585.759} C_VEL
LIN {X 0,Y 200.012,Z 281.064,A -85,B 0,C 180,E1 -21589.894,E2 -21589.894} C_VEL
LIN {X 0,Y 200.001,Z 281.071,A -85,B 0,C 180,E1 -21593.961,E2 -21593.961} C_VEL
LIN {X 0,Y 200.284,Z 281.006,A -85,B 0,C 180,E1 -21598.001,E2 -21598.001} C_VEL
LIN {X 0,Y 200.442,Z 281,A -85,B 0,C 180,E1 -21600.012,E2 -21600.012} C_VEL
LIN {X 0,Y 199.985,Z 281.074,A -85,B 0,C 180,E1 -21604.042,E2 -21604.042} C_VEL
LIN {X 0,Y 200.076,Z 281.064,A -85,B 0,C 180,E1 -21608.088,E2 -21608.088} C_VEL
LIN {X 0,Y 199.857,Z 281.092,A -85,B 0,C 180,E1 -21612.192,E2 -21612.192} C_VEL
LIN {X 0,Y 199.749,Z 281.104,A -85,B 0,C 180,E1 -21616.359,E2 -21616.359} C_VEL
LIN {X 0,Y 199.65,Z 281.116,A -85,B 0,C 180,E1 -21620.622,E2 -21620.622} C_VEL
LIN {X 0,Y 199.64,Z 281.146,A -85,B 0,C 180,E1 -21625,E2 -21625} C_VEL
LIN {X 0,Y 199.829,Z 282.704,A -85,B 0,C 180,E1 -21629.509,E2 -21629.509} C_VEL
LIN {X 0,Y 200.113,Z 284.567,A -85,B 0,C 180,E1 -21634.201,E2 -21634.201} C_VEL
LIN {X 0,Y 200.452,Z 286.961,A -85,B 0,C 180,E1 -21639.527,E2 -21639.527} C_VEL
LIN {X 0,Y 200.661,Z 288.503,A -85,B 0,C 180,E1 -21642.651,E2 -21642.651} C_VEL
LIN {X 0,Y 200.728,Z 290.036,A -85,B 0,C 180,E1 -21645.554,E2 -21645.554} C_VEL
LIN {X 0,Y 200.587,Z 291.565,A -85,B 0,C 180,E1 -21648.264,E2 -21648.264} C_VEL
LIN {X 0,Y 200.083,Z 293.795,A -85,B 0,C 180,E1 -21651.848,E2 -21651.848} C_VEL
LIN {X 0,Y 200.971,Z 296.993,A -85,B 0,C 180,E1 -21652.237,E2 -21652.237} C_VEL
LIN {X 0,Y 201.964,Z 299.498,A -85,B 0,C 180,E1 -21652.641,E2 -21652.641} C_VEL
LIN {X 0,Y 205.76,Z 311.018,A -85,B 0,C 180,E1 -21654.504,E2 -21654.504} C_VEL
LIN {X 0,Y 208.199,Z 321.311,A -85,B 0,C 180,E1 -21656.227,E2 -21656.227} C_VEL
LIN {X 0,Y 209.748,Z 330.909,A -85,B 0,C 180,E1 -21657.946,E2 -21657.946} C_VEL
LIN {X 0,Y 210.575,Z 340.038,A -85,B 0,C 180,E1 -21659.727,E2 -21659.727} C_VEL
LIN {X 0,Y 210.795,Z 347.603,A -85,B 0,C 180,E1 -21661.339,E2 -21661.339} C_VEL
LIN {X 0,Y 210.333,Z 355.508,A -85,B 0,C 180,E1 -21663.187,E2 -21663.187} C_VEL
LIN {X 0,Y 207.475,Z 364.644,A -85,B 0,C 180,E1 -21665.484,E2 -21665.484} C_VEL
LIN {X 0,Y 205.145,Z 372.228,A -85,B 0,C 180,E1 -21667.862,E2 -21667.862} C_VEL
LIN {X 0,Y 203.433,Z 377.391,A -85,B 0,C 180,E1 -21669.79,E2 -21669.79} C_VEL
LIN {X 0,Y 201.966,Z 381.896,A -85,B 0,C 180,E1 -21671.749,E2 -21671.749} C_VEL
LIN {X 0,Y 200.024,Z 387.389,A -85,B 0,C 180,E1 -21674.721,E2 -21674.721} C_VEL
LIN {X 0,Y 198.689,Z 391.72,A -85,B 0,C 180,E1 -21677.747,E2 -21677.747} C_VEL
LIN {X 0,Y 197.913,Z 394.642,A -85,B 0,C 180,E1 -21680.401,E2 -21680.401} C_VEL
LIN {X 0,Y 197.377,Z 397.291,A -85,B 0,C 180,E1 -21683.868,E2 -21683.868} C_VEL
LIN {X 0,Y 197.268,Z 398.412,A -85,B 0,C 180,E1 -21686.107,E2 -21686.107} C_VEL
LIN {X 0,Y 197.279,Z 399.044,A -85,B 0,C 180,E1 -21689.183,E2 -21689.183} C_VEL
LIN {X 0,Y 196.656,Z 399.11,A -85,B 0,C 180,E1 -21690.885,E2 -21690.885} C_VEL
LIN {X 0,Y 195.069,Z 398.793,A -85,B 0,C 180,E1 -21692.557,E2 -21692.557} C_VEL
LIN {X 0,Y 191.408,Z 397.339,A -85,B 0,C 180,E1 -21695.923,E2 -21695.923} C_VEL
LIN {X 0,Y 190.518,Z 396.121,A -85,B 0,C 180,E1 -21697.966,E2 -21697.966} C_VEL
LIN {X 0,Y 190.545,Z 395.831,A -85,B 0,C 180,E1 -21698.261,E2 -21698.261} C_VEL
LIN {X 0,Y 191.361,Z 392.728,A -85,B 0,C 180,E1 -21701.653,E2 -21701.653} C_VEL
LIN {X 0,Y 192.572,Z 388.731,A -85,B 0,C 180,E1 -21704.801,E2 -21704.801} C_VEL
LIN {X 0,Y 194.444,Z 383.6,A -85,B 0,C 180,E1 -21707.892,E2 -21707.892} C_VEL
LIN {X 0,Y 196.31,Z 378.334,A -85,B 0,C 180,E1 -21710.429,E2 -21710.429} C_VEL
LIN {X 0,Y 198.112,Z 373.416,A -85,B 0,C 180,E1 -21712.408,E2 -21712.408} C_VEL
LIN {X 0,Y 200.464,Z 366.059,A -85,B 0,C 180,E1 -21714.879,E2 -21714.879} C_VEL
LIN {X 0,Y 202.706,Z 359.132,A -85,B 0,C 180,E1 -21716.789,E2 -21716.789} C_VEL
LIN {X 0,Y 203.979,Z 354.302,A -85,B 0,C 180,E1 -21717.998,E2 -21717.998} C_VEL
LIN {X 0,Y 204.228,Z 344.752,A -85,B 0,C 180,E1 -21720.28,E2 -21720.28} C_VEL
LIN {X 0,Y 203.603,Z 334.462,A -85,B 0,C 180,E1 -21722.469,E2 -21722.469} C_VEL
LIN {X 0,Y 202.484,Z 325.723,A -85,B 0,C 180,E1 -21724.175,E2 -21724.175} C_VEL
LIN {X 0,Y 200.21,Z 314.895,A -85,B 0,C 180,E1 -21726.145,E2 -21726.145} C_VEL
LIN {X 0,Y 197.271,Z 304.925,A -85,B 0,C 180,E1 -21727.889,E2 -21727.889} C_VEL
LIN {X 0,Y 194.598,Z 297.473,A -85,B 0,C 180,E1 -21729.183,E2 -21729.183} C_VEL
LIN {X 0,Y 193.466,Z 294.711,A -85,B 0,C 180,E1 -21729.632,E2 -21729.632} C_VEL
LIN {X 0,Y 193.282,Z 293.537,A -85,B 0,C 180,E1 -21729.78,E2 -21729.78} C_VEL
LIN {X 0,Y 193.618,Z 291.322,A -85,B 0,C 180,E1 -21733.603,E2 -21733.603} C_VEL
LIN {X 0,Y 193.612,Z 289.768,A -85,B 0,C 180,E1 -21736.55,E2 -21736.55} C_VEL
LIN {X 0,Y 193.459,Z 288.246,A -85,B 0,C 180,E1 -21739.718,E2 -21739.718} C_VEL
LIN {X 0,Y 193.141,Z 286.189,A -85,B 0,C 180,E1 -21744.382,E2 -21744.382} C_VEL
LIN {X 0,Y 193.032,Z 285.165,A -85,B 0,C 180,E1 -21746.886,E2 -21746.886} C_VEL
LIN {X 0,Y 192.78,Z 283.364,A -85,B 0,C 180,E1 -21751.699,E2 -21751.699} C_VEL
LIN {X 0,Y 192.656,Z 281.994,A -85,B 0,C 180,E1 -21756.33,E2 -21756.33} C_VEL
LIN {X 0,Y 192.703,Z 281.984,A -85,B 0,C 180,E1 -21761.481,E2 -21761.481} C_VEL
LIN {X 0,Y 192.779,Z 281.971,A -85,B 0,C 180,E1 -21767.353,E2 -21767.353} C_VEL
LIN {X 0,Y 193.027,Z 281.941,A -85,B 0,C 180,E1 -21771.614,E2 -21771.614} C_VEL
LIN {X 0,Y 193.227,Z 281.913,A -85,B 0,C 180,E1 -21777.904,E2 -21777.904} C_VEL
LIN {X 0,Y 193.409,Z 281.876,A -85,B 0,C 180,E1 -21779.988,E2 -21779.988} C_VEL
LIN {X 0,Y 192.938,Z 281.933,A -85,B 0,C 180,E1 -21784.165,E2 -21784.165} C_VEL
LIN {X 0,Y 193.019,Z 281.939,A -85,B 0,C 180,E1 -21788.362,E2 -21788.362} C_VEL
LIN {X 0,Y 192.779,Z 281.971,A -85,B 0,C 180,E1 -21792.622,E2 -21792.622} C_VEL
LIN {X 0,Y 192.703,Z 281.98,A -85,B 0,C 180,E1 -21796.95,E2 -21796.95} C_VEL
LIN {X 0,Y 192.584,Z 281.993,A -85,B 0,C 180,E1 -21801.389,E2 -21801.389} C_VEL
LIN {X 0,Y 192.625,Z 281.986,A -85,B 0,C 180,E1 -21804.201,E2 -21804.201} C_VEL
LIN {X 0,Y 192.625,Z 281.99,A -85,B 0,C 180,E1 -21808.88,E2 -21808.88} C_VEL
LIN {X 0,Y 192.572,Z 281.996,A -85,B 0,C 180,E1 -21813.174,E2 -21813.174} C_VEL
LIN {X 0,Y 192.569,Z 281.997,A -85,B 0,C 180,E1 -21818.329,E2 -21818.329} C_VEL
LIN {X 0,Y 192.577,Z 281.996,A -85,B 0,C 180,E1 -21823.124,E2 -21823.124} C_VEL
LIN {X 0,Y 192.574,Z 281.996,A -85,B 0,C 180,E1 -21826.856,E2 -21826.856} C_VEL
LIN {X 0,Y 192.558,Z 281.998,A -85,B 0,C 180,E1 -21829.854,E2 -21829.854} C_VEL
LIN {X 0,Y 193.668,Z 284.996,A -85,B 0,C 180,E1 -21830.364,E2 -21830.364} C_VEL
LIN {X 0,Y 195.241,Z 287.045,A -85,B 0,C 180,E1 -21830.878,E2 -21830.878} C_VEL
LIN {X 0,Y 201.501,Z 298.495,A -85,B 0,C 180,E1 -21833.317,E2 -21833.317} C_VEL
LIN {X 0,Y 206.469,Z 309.452,A -85,B 0,C 180,E1 -21835.662,E2 -21835.662} C_VEL
LIN {X 0,Y 210.221,Z 319.752,A -85,B 0,C 180,E1 -21837.923,E2 -21837.923} C_VEL
LIN {X 0,Y 212.893,Z 328.89,A -85,B 0,C 180,E1 -21840.033,E2 -21840.033} C_VEL
LIN {X 0,Y 215.771,Z 336.851,A -85,B 0,C 180,E1 -21842.15,E2 -21842.15} C_VEL
LIN {X 0,Y 220.237,Z 345.571,A -85,B 0,C 180,E1 -21844.89,E2 -21844.89} C_VEL
LIN {X 0,Y 225.237,Z 352.786,A -85,B 0,C 180,E1 -21847.501,E2 -21847.501} C_VEL
LIN {X 0,Y 231.98,Z 360.111,A -85,B 0,C 180,E1 -21850.534,E2 -21850.534} C_VEL
LIN {X 0,Y 238.754,Z 365.899,A -85,B 0,C 180,E1 -21853.243,E2 -21853.243} C_VEL
LIN {X 0,Y 246.22,Z 371.099,A -85,B 0,C 180,E1 -21855.99,E2 -21855.99} C_VEL
LIN {X 0,Y 254.375,Z 375.805,A -85,B 0,C 180,E1 -21858.849,E2 -21858.849} C_VEL
LIN {X 0,Y 259.46,Z 378.381,A -85,B 0,C 180,E1 -21860.647,E2 -21860.647} C_VEL
LIN {X 0,Y 263.983,Z 380.501,A -85,B 0,C 180,E1 -21862.351,E2 -21862.351} C_VEL
LIN {X 0,Y 268.375,Z 382.395,A -85,B 0,C 180,E1 -21864.211,E2 -21864.211} C_VEL
LIN {X 0,Y 270.721,Z 383.466,A -85,B 0,C 180,E1 -21865.533,E2 -21865.533} C_VEL
LIN {X 0,Y 274.217,Z 384.731,A -85,B 0,C 180,E1 -21867.906,E2 -21867.906} C_VEL
LIN {X 0,Y 274.959,Z 384.927,A -85,B 0,C 180,E1 -21868.535,E2 -21868.535} C_VEL
LIN {X 0,Y 276.209,Z 385.082,A -85,B 0,C 180,E1 -21870,E2 -21870} C_VEL
LIN {X 0,Y 274.215,Z 384.735,A -85,B 0,C 180,E1 -21872.081,E2 -21872.081} C_VEL
LIN {X 0,Y 270.72,Z 383.466,A -85,B 0,C 180,E1 -21874.467,E2 -21874.467} C_VEL
LIN {X 0,Y 267.82,Z 382.182,A -85,B 0,C 180,E1 -21876.025,E2 -21876.025} C_VEL
LIN {X 0,Y 262.651,Z 379.871,A -85,B 0,C 180,E1 -21878.179,E2 -21878.179} C_VEL
LIN {X 0,Y 257.036,Z 377.183,A -85,B 0,C 180,E1 -21880.228,E2 -21880.228} C_VEL
LIN {X 0,Y 248.94,Z 372.791,A -85,B 0,C 180,E1 -21883.053,E2 -21883.053} C_VEL
LIN {X 0,Y 241.079,Z 367.648,A -85,B 0,C 180,E1 -21885.889,E2 -21885.889} C_VEL
LIN {X 0,Y 233.726,Z 361.738,A -85,B 0,C 180,E1 -21888.749,E2 -21888.749} C_VEL
LIN {X 0,Y 226.609,Z 354.433,A -85,B 0,C 180,E1 -21891.849,E2 -21891.849} C_VEL
LIN {X 0,Y 221.61,Z 347.782,A -85,B 0,C 180,E1 -21894.347,E2 -21894.347} C_VEL
LIN {X 0,Y 217.19,Z 339.872,A -85,B 0,C 180,E1 -21896.937,E2 -21896.937} C_VEL
LIN {X 0,Y 213.668,Z 331.16,A -85,B 0,C 180,E1 -21899.381,E2 -21899.381} C_VEL
LIN {X 0,Y 211.036,Z 322.546,A -85,B 0,C 180,E1 -21901.448,E2 -21901.448} C_VEL
LIN {X 0,Y 208.334,Z 314.201,A -85,B 0,C 180,E1 -21903.288,E2 -21903.288} C_VEL
LIN {X 0,Y 204.481,Z 304.845,A -85,B 0,C 180,E1 -21905.311,E2 -21905.311} C_VEL
LIN {X 0,Y 199.746,Z 295.202,A -85,B 0,C 180,E1 -21907.373,E2 -21907.373} C_VEL
LIN {X 0,Y 194.517,Z 286.023,A -85,B 0,C 180,E1 -21909.38,E2 -21909.38} C_VEL
LIN {X 0,Y 192.938,Z 283.578,A -85,B 0,C 180,E1 -21909.935,E2 -21909.935} C_VEL
LIN {X 0,Y 192.558,Z 281.998,A -85,B 0,C 180,E1 -21910.146,E2 -21910.146} C_VEL
LIN {X 0,Y 192.583,Z 281.997,A -85,B 0,C 180,E1 -21913.897,E2 -21913.897} C_VEL
LIN {X 0,Y 192.577,Z 281.996,A -85,B 0,C 180,E1 -21916.876,E2 -21916.876} C_VEL
LIN {X 0,Y 192.569,Z 281.997,A -85,B 0,C 180,E1 -21921.671,E2 -21921.671} C_VEL
LIN {X 0,Y 192.572,Z 281.996,A -85,B 0,C 180,E1 -21926.826,E2 -21926.826} C_VEL
LIN {X 0,Y 192.64,Z 281.989,A -85,B 0,C 180,E1 -21931.704,E2 -21931.704} C_VEL
LIN {X 0,Y 192.663,Z 281.983,A -85,B 0,C 180,E1 -21936.358,E2 -21936.358} C_VEL
LIN {X 0,Y 192.681,Z 281.983,A -85,B 0,C 180,E1 -21941.501,E2 -21941.501} C_VEL
LIN {X 0,Y 192.724,Z 281.971,A -85,B 0,C 180,E1 -21945.224,E2 -21945.224} C_VEL
LIN {X 0,Y 192.935,Z 281.946,A -85,B 0,C 180,E1 -21949.579,E2 -21949.579} C_VEL
LIN {X 0,Y 192.964,Z 281.948,A -85,B 0,C 180,E1 -21953.74,E2 -21953.74} C_VEL
LIN {X 0,Y 193.229,Z 281.883,A -85,B 0,C 180,E1 -21957.928,E2 -21957.928} C_VEL
LIN {X 0,Y 193.409,Z 281.876,A -85,B 0,C 180,E1 -21960.012,E2 -21960.012} C_VEL
LIN {X 0,Y 192.933,Z 281.953,A -85,B 0,C 180,E1 -21964.19,E2 -21964.19} C_VEL
LIN {X 0,Y 193.027,Z 281.941,A -85,B 0,C 180,E1 -21968.386,E2 -21968.386} C_VEL
LIN {X 0,Y 192.779,Z 281.972,A -85,B 0,C 180,E1 -21972.647,E2 -21972.647} C_VEL
LIN {X 0,Y 192.703,Z 281.982,A -85,B 0,C 180,E1 -21978.519,E2 -21978.519} C_VEL
LIN {X 0,Y 192.623,Z 282.014,A -85,B 0,C 180,E1 -21984.199,E2 -21984.199} C_VEL
LIN {X 0,Y 192.796,Z 283.602,A -85,B 0,C 180,E1 -21988.972,E2 -21988.972} C_VEL
LIN {X 0,Y 193.02,Z 285.172,A -85,B 0,C 180,E1 -21993.13,E2 -21993.13} C_VEL
LIN {X 0,Y 193.286,Z 287.299,A -85,B 0,C 180,E1 -21998.192,E2 -21998.192} C_VEL
LIN {X 0,Y 193.498,Z 288.531,A -85,B 0,C 180,E1 -22000.84,E2 -22000.84} C_VEL
LIN {X 0,Y 193.653,Z 289.889,A -85,B 0,C 180,E1 -22003.607,E2 -22003.607} C_VEL
LIN {X 0,Y 193.622,Z 291.428,A -85,B 0,C 180,E1 -22006.562,E2 -22006.562} C_VEL
LIN {X 0,Y 193.279,Z 293.511,A -85,B 0,C 180,E1 -22010.22,E2 -22010.22} C_VEL
LIN {X 0,Y 194.292,Z 296.948,A -85,B 0,C 180,E1 -22010.708,E2 -22010.708} C_VEL
LIN {X 0,Y 195.098,Z 298.743,A -85,B 0,C 180,E1 -22011.039,E2 -22011.039} C_VEL
LIN {X 0,Y 199.09,Z 310.772,A -85,B 0,C 180,E1 -22013.123,E2 -22013.123} C_VEL
LIN {X 0,Y 201.575,Z 320.887,A -85,B 0,C 180,E1 -22014.931,E2 -22014.931} C_VEL
LIN {X 0,Y 203.242,Z 331.004,A -85,B 0,C 180,E1 -22016.849,E2 -22016.849} C_VEL
LIN {X 0,Y 204.014,Z 339.95,A -85,B 0,C 180,E1 -22018.675,E2 -22018.675} C_VEL
LIN {X 0,Y 204.243,Z 347.921,A -85,B 0,C 180,E1 -22020.463,E2 -22020.463} C_VEL
LIN {X 0,Y 203.903,Z 355.292,A -85,B 0,C 180,E1 -22022.27,E2 -22022.27} C_VEL
LIN {X 0,Y 201.011,Z 364.432,A -85,B 0,C 180,E1 -22024.641,E2 -22024.641} C_VEL
LIN {X 0,Y 198.674,Z 371.535,A -85,B 0,C 180,E1 -22026.909,E2 -22026.909} C_VEL
LIN {X 0,Y 196.78,Z 377.18,A -85,B 0,C 180,E1 -22029.075,E2 -22029.075} C_VEL
LIN {X 0,Y 195.198,Z 381.684,A -85,B 0,C 180,E1 -22031.093,E2 -22031.093} C_VEL
LIN {X 0,Y 193.144,Z 387.177,A -85,B 0,C 180,E1 -22034.163,E2 -22034.163} C_VEL
LIN {X 0,Y 191.73,Z 391.508,A -85,B 0,C 180,E1 -22037.295,E2 -22037.295} C_VEL
LIN {X 0,Y 191.068,Z 393.881,A -85,B 0,C 180,E1 -22039.402,E2 -22039.402} C_VEL
LIN {X 0,Y 190.313,Z 397.079,A -85,B 0,C 180,E1 -22043.639,E2 -22043.639} C_VEL
LIN {X 0,Y 190.177,Z 398.301,A -85,B 0,C 180,E1 -22046.32,E2 -22046.32} C_VEL
LIN {X 0,Y 190.248,Z 398.897,A -85,B 0,C 180,E1 -22050,E2 -22050} C_VEL
LIN {X 0,Y 190.154,Z 398.331,A -85,B 0,C 180,E1 -22053.571,E2 -22053.571} C_VEL
LIN {X 0,Y 190.324,Z 397.08,A -85,B 0,C 180,E1 -22056.36,E2 -22056.36} C_VEL
LIN {X 0,Y 190.545,Z 395.831,A -85,B 0,C 180,E1 -22058.261,E2 -22058.261} C_VEL
LIN {X 0,Y 190.228,Z 394.509,A -85,B 0,C 180,E1 -22059.99,E2 -22059.99} C_VEL
LIN {X 0,Y 188.179,Z 391.672,A -85,B 0,C 180,E1 -22062.801,E2 -22062.801} C_VEL
LIN {X 0,Y 186.687,Z 388.888,A -85,B 0,C 180,E1 -22065.04,E2 -22065.04} C_VEL
LIN {X 0,Y 186.543,Z 386.557,A -85,B 0,C 180,E1 -22066.709,E2 -22066.709} C_VEL
LIN {X 0,Y 186.798,Z 385.689,A -85,B 0,C 180,E1 -22067.254,E2 -22067.254} C_VEL
LIN {X 0,Y 189.207,Z 379.278,A -85,B 0,C 180,E1 -22070.663,E2 -22070.663} C_VEL
LIN {X 0,Y 191.555,Z 373.117,A -85,B 0,C 180,E1 -22073.255,E2 -22073.255} C_VEL
LIN {X 0,Y 193.469,Z 367.474,A -85,B 0,C 180,E1 -22075.266,E2 -22075.266} C_VEL
LIN {X 0,Y 196.393,Z 358.921,A -85,B 0,C 180,E1 -22077.723,E2 -22077.723} C_VEL
LIN {X 0,Y 197.371,Z 355.072,A -85,B 0,C 180,E1 -22078.731,E2 -22078.731} C_VEL
LIN {X 0,Y 197.746,Z 345.806,A -85,B 0,C 180,E1 -22081.092,E2 -22081.092} C_VEL
LIN {X 0,Y 197.124,Z 334.696,A -85,B 0,C 180,E1 -22083.589,E2 -22083.589} C_VEL
LIN {X 0,Y 195.821,Z 324.97,A -85,B 0,C 180,E1 -22085.589,E2 -22085.589} C_VEL
LIN {X 0,Y 193.752,Z 315.026,A -85,B 0,C 180,E1 -22087.506,E2 -22087.506} C_VEL
LIN {X 0,Y 190.489,Z 304.45,A -85,B 0,C 180,E1 -22089.515,E2 -22089.515} C_VEL
LIN {X 0,Y 187.991,Z 297.593,A -85,B 0,C 180,E1 -22090.814,E2 -22090.814} C_VEL
LIN {X 0,Y 186.588,Z 294.569,A -85,B 0,C 180,E1 -22091.396,E2 -22091.396} C_VEL
LIN {X 0,Y 186.385,Z 293.282,A -85,B 0,C 180,E1 -22091.584,E2 -22091.584} C_VEL
LIN {X 0,Y 186.536,Z 291.066,A -85,B 0,C 180,E1 -22095.712,E2 -22095.712} C_VEL
LIN {X 0,Y 186.393,Z 288.991,A -85,B 0,C 180,E1 -22100.121,E2 -22100.121} C_VEL
LIN {X 0,Y 186.033,Z 286.748,A -85,B 0,C 180,E1 -22105.469,E2 -22105.469} C_VEL
LIN {X 0,Y 185.787,Z 284.881,A -85,B 0,C 180,E1 -22110.531,E2 -22110.531} C_VEL
LIN {X 0,Y 185.6,Z 283.293,A -85,B 0,C 180,E1 -22115.372,E2 -22115.372} C_VEL
LIN {X 0,Y 185.549,Z 282.879,A -85,B 0,C 180,E1 -22117.73,E2 -22117.73} C_VEL
LIN {X 0,Y 185.654,Z 282.862,A -85,B 0,C 180,E1 -22122.359,E2 -22122.359} C_VEL
LIN {X 0,Y 185.704,Z 282.853,A -85,B 0,C 180,E1 -22126.863,E2 -22126.863} C_VEL
LIN {X 0,Y 185.977,Z 282.819,A -85,B 0,C 180,E1 -22131.294,E2 -22131.294} C_VEL
LIN {X 0,Y 186.173,Z 282.792,A -85,B 0,C 180,E1 -22137.824,E2 -22137.824} C_VEL
LIN {X 0,Y 186.375,Z 282.75,A -85,B 0,C 180,E1 -22139.987,E2 -22139.987} C_VEL
LIN {X 0,Y 185.886,Z 282.812,A -85,B 0,C 180,E1 -22144.324,E2 -22144.324} C_VEL
LIN {X 0,Y 185.968,Z 282.817,A -85,B 0,C 180,E1 -22148.681,E2 -22148.681} C_VEL
LIN {X 0,Y 185.704,Z 282.852,A -85,B 0,C 180,E1 -22153.111,E2 -22153.111} C_VEL
LIN {X 0,Y 185.639,Z 282.861,A -85,B 0,C 180,E1 -22157.616,E2 -22157.616} C_VEL
LIN {X 0,Y 185.551,Z 282.872,A -85,B 0,C 180,E1 -22162.242,E2 -22162.242} C_VEL
LIN {X 0,Y 185.537,Z 282.874,A -85,B 0,C 180,E1 -22167.02,E2 -22167.02} C_VEL
LIN {X 0,Y 185.554,Z 282.872,A -85,B 0,C 180,E1 -22169.481,E2 -22169.481} C_VEL
LIN {X 0,Y 185.492,Z 282.88,A -85,B 0,C 180,E1 -22174.616,E2 -22174.616} C_VEL
LIN {X 0,Y 185.537,Z 282.874,A -85,B 0,C 180,E1 -22177.303,E2 -22177.303} C_VEL
LIN {X 0,Y 185.529,Z 282.874,A -85,B 0,C 180,E1 -22180.747,E2 -22180.747} C_VEL
LIN {X 0,Y 185.542,Z 282.874,A -85,B 0,C 180,E1 -22186.007,E2 -22186.007} C_VEL
LIN {X 0,Y 185.529,Z 283.039,A -85,B 0,C 180,E1 -22188.093,E2 -22188.093} C_VEL
LIN {X 0,Y 186.453,Z 285.615,A -85,B 0,C 180,E1 -22188.525,E2 -22188.525} C_VEL
LIN {X 0,Y 188.3,Z 288.046,A -85,B 0,C 180,E1 -22189.187,E2 -22189.187} C_VEL
LIN {X 0,Y 194.485,Z 298.987,A -85,B 0,C 180,E1 -22191.786,E2 -22191.786} C_VEL
LIN {X 0,Y 199.868,Z 310.688,A -85,B 0,C 180,E1 -22194.515,E2 -22194.515} C_VEL
LIN {X 0,Y 203.501,Z 320.62,A -85,B 0,C 180,E1 -22196.847,E2 -22196.847} C_VEL
LIN {X 0,Y 206.266,Z 330.509,A -85,B 0,C 180,E1 -22199.264,E2 -22199.264} C_VEL
LIN {X 0,Y 208.991,Z 338.798,A -85,B 0,C 180,E1 -22201.587,E2 -22201.587} C_VEL
LIN {X 0,Y 212.278,Z 345.85,A -85,B 0,C 180,E1 -22203.886,E2 -22203.886} C_VEL
LIN {X 0,Y 216.808,Z 353.1,A -85,B 0,C 180,E1 -22206.591,E2 -22206.591} C_VEL
LIN {X 0,Y 222.981,Z 360.389,A -85,B 0,C 180,E1 -22209.715,E2 -22209.715} C_VEL
LIN {X 0,Y 228.716,Z 365.599,A -85,B 0,C 180,E1 -22212.238,E2 -22212.238} C_VEL
LIN {X 0,Y 236.192,Z 371.003,A -85,B 0,C 180,E1 -22215.196,E2 -22215.196} C_VEL
LIN {X 0,Y 245.044,Z 376.085,A -85,B 0,C 180,E1 -22218.419,E2 -22218.419} C_VEL
LIN {X 0,Y 252.881,Z 379.75,A -85,B 0,C 180,E1 -22221.208,E2 -22221.208} C_VEL
LIN {X 0,Y 255.36,Z 380.801,A -85,B 0,C 180,E1 -22222.124,E2 -22222.124} C_VEL
LIN {X 0,Y 261.182,Z 383.057,A -85,B 0,C 180,E1 -22224.498,E2 -22224.498} C_VEL
LIN {X 0,Y 262.908,Z 383.698,A -85,B 0,C 180,E1 -22225.4,E2 -22225.4} C_VEL
LIN {X 0,Y 265.411,Z 384.628,A -85,B 0,C 180,E1 -22226.964,E2 -22226.964} C_VEL
LIN {X 0,Y 267.608,Z 385.145,A -85,B 0,C 180,E1 -22228.495,E2 -22228.495} C_VEL
LIN {X 0,Y 268.993,Z 385.293,A -85,B 0,C 180,E1 -22230,E2 -22230} C_VEL
LIN {X 0,Y 267.144,Z 385.047,A -85,B 0,C 180,E1 -22231.837,E2 -22231.837} C_VEL
LIN {X 0,Y 265.392,Z 384.628,A -85,B 0,C 180,E1 -22233.036,E2 -22233.036} C_VEL
LIN {X 0,Y 262.907,Z 383.697,A -85,B 0,C 180,E1 -22234.6,E2 -22234.6} C_VEL
LIN {X 0,Y 261.182,Z 383.057,A -85,B 0,C 180,E1 -22235.502,E2 -22235.502} C_VEL
LIN {X 0,Y 255.26,Z 380.763,A -85,B 0,C 180,E1 -22237.913,E2 -22237.913} C_VEL
LIN {X 0,Y 247.699,Z 377.405,A -85,B 0,C 180,E1 -22240.657,E2 -22240.657} C_VEL
LIN {X 0,Y 238.805,Z 372.641,A -85,B 0,C 180,E1 -22243.843,E2 -22243.843} C_VEL
LIN {X 0,Y 231.171,Z 367.483,A -85,B 0,C 180,E1 -22246.78,E2 -22246.78} C_VEL
LIN {X 0,Y 224.053,Z 361.397,A -85,B 0,C 180,E1 -22249.816,E2 -22249.816} C_VEL
LIN {X 0,Y 217.981,Z 354.703,A -85,B 0,C 180,E1 -22252.761,E2 -22252.761} C_VEL
LIN {X 0,Y 213.08,Z 347.275,A -85,B 0,C 180,E1 -22255.605,E2 -22255.605} C_VEL
LIN {X 0,Y 209.568,Z 340.119,A -85,B 0,C 180,E1 -22258.001,E2 -22258.001} C_VEL
LIN {X 0,Y 206.623,Z 331.83,A -85,B 0,C 180,E1 -22260.394,E2 -22260.394} C_VEL
LIN {X 0,Y 204.219,Z 323.161,A -85,B 0,C 180,E1 -22262.555,E2 -22262.555} C_VEL
LIN {X 0,Y 201.583,Z 315.256,A -85,B 0,C 180,E1 -22264.432,E2 -22264.432} C_VEL
LIN {X 0,Y 197.392,Z 305.013,A -85,B 0,C 180,E1 -22266.791,E2 -22266.791} C_VEL
LIN {X 0,Y 192.384,Z 295.111,A -85,B 0,C 180,E1 -22269.102,E2 -22269.102} C_VEL
LIN {X 0,Y 189.625,Z 290.511,A -85,B 0,C 180,E1 -22270.252,E2 -22270.252} C_VEL
LIN {X 0,Y 187.692,Z 287.161,A -85,B 0,C 180,E1 -22271.047,E2 -22271.047} C_VEL
LIN {X 0,Y 185.988,Z 284.713,A -85,B 0,C 180,E1 -22271.69,E2 -22271.69} C_VEL
LIN {X 0,Y 185.498,Z 282.878,A -85,B 0,C 180,E1 -22271.971,E2 -22271.971} C_VEL
LIN {X 0,Y 185.543,Z 282.874,A -85,B 0,C 180,E1 -22276.027,E2 -22276.027} C_VEL
LIN {X 0,Y 185.509,Z 282.877,A -85,B 0,C 180,E1 -22279.925,E2 -22279.925} C_VEL
LIN {X 0,Y 185.529,Z 282.875,A -85,B 0,C 180,E1 -22282.711,E2 -22282.711} C_VEL
LIN {X 0,Y 185.518,Z 282.876,A -85,B 0,C 180,E1 -22287.987,E2 -22287.987} C_VEL
LIN {X 0,Y 185.557,Z 282.872,A -85,B 0,C 180,E1 -22290.588,E2 -22290.588} C_VEL
LIN {X 0,Y 185.559,Z 282.864,A -85,B 0,C 180,E1 -22295.394,E2 -22295.394} C_VEL
LIN {X 0,Y 185.611,Z 282.861,A -85,B 0,C 180,E1 -22301.189,E2 -22301.189} C_VEL
LIN {X 0,Y 185.653,Z 282.852,A -85,B 0,C 180,E1 -22304.648,E2 -22304.648} C_VEL
LIN {X 0,Y 185.878,Z 282.826,A -85,B 0,C 180,E1 -22309.432,E2 -22309.432} C_VEL
LIN {X 0,Y 185.928,Z 282.824,A -85,B 0,C 180,E1 -22313.502,E2 -22313.502} C_VEL
LIN {X 0,Y 186.175,Z 282.76,A -85,B 0,C 180,E1 -22317.849,E2 -22317.849} C_VEL
LIN {X 0,Y 186.375,Z 282.75,A -85,B 0,C 180,E1 -22320.013,E2 -22320.013} C_VEL
LIN {X 0,Y 185.881,Z 282.831,A -85,B 0,C 180,E1 -22324.349,E2 -22324.349} C_VEL
LIN {X 0,Y 185.977,Z 282.819,A -85,B 0,C 180,E1 -22328.706,E2 -22328.706} C_VEL
LIN {X 0,Y 185.704,Z 282.854,A -85,B 0,C 180,E1 -22333.137,E2 -22333.137} C_VEL
LIN {X 0,Y 185.634,Z 282.862,A -85,B 0,C 180,E1 -22338.832,E2 -22338.832} C_VEL
LIN {X 0,Y 185.549,Z 282.872,A -85,B 0,C 180,E1 -22342.27,E2 -22342.27} C_VEL
LIN {X 0,Y 185.631,Z 283.301,A -85,B 0,C 180,E1 -22344.684,E2 -22344.684} C_VEL
LIN {X 0,Y 185.78,Z 284.902,A -85,B 0,C 180,E1 -22349.533,E2 -22349.533} C_VEL
LIN {X 0,Y 186.038,Z 286.745,A -85,B 0,C 180,E1 -22354.53,E2 -22354.53} C_VEL
LIN {X 0,Y 186.393,Z 289,A -85,B 0,C 180,E1 -22359.879,E2 -22359.879} C_VEL
LIN {X 0,Y 186.562,Z 291.09,A -85,B 0,C 180,E1 -22364.296,E2 -22364.296} C_VEL
LIN {X 0,Y 186.375,Z 293.271,A -85,B 0,C 180,E1 -22368.42,E2 -22368.42} C_VEL
LIN {X 0,Y 187.234,Z 296.279,A -85,B 0,C 180,E1 -22368.891,E2 -22368.891} C_VEL
LIN {X 0,Y 188.568,Z 299.082,A -85,B 0,C 180,E1 -22369.475,E2 -22369.475} C_VEL
LIN {X 0,Y 192.222,Z 309.612,A -85,B 0,C 180,E1 -22371.455,E2 -22371.455} C_VEL
LIN {X 0,Y 194.994,Z 320.471,A -85,B 0,C 180,E1 -22373.534,E2 -22373.534} C_VEL
LIN {X 0,Y 196.575,Z 329.501,A -85,B 0,C 180,E1 -22375.332,E2 -22375.332} C_VEL
LIN {X 0,Y 197.466,Z 339.009,A -85,B 0,C 180,E1 -22377.354,E2 -22377.354} C_VEL
LIN {X 0,Y 197.726,Z 348.257,A -85,B 0,C 180,E1 -22379.532,E2 -22379.532} C_VEL
LIN {X 0,Y 197.376,Z 355.072,A -85,B 0,C 180,E1 -22381.27,E2 -22381.27} C_VEL
LIN {X 0,Y 196.425,Z 358.922,A -85,B 0,C 180,E1 -22382.282,E2 -22382.282} C_VEL
LIN {X 0,Y 193.476,Z 367.475,A -85,B 0,C 180,E1 -22384.735,E2 -22384.735} C_VEL
LIN {X 0,Y 190.587,Z 375.974,A -85,B 0,C 180,E1 -22387.872,E2 -22387.872} C_VEL
LIN {X 0,Y 188.457,Z 381.471,A -85,B 0,C 180,E1 -22390.389,E2 -22390.389} C_VEL
LIN {X 0,Y 186.295,Z 386.965,A -85,B 0,C 180,E1 -22393.565,E2 -22393.565} C_VEL
LIN {X 0,Y 184.787,Z 391.296,A -85,B 0,C 180,E1 -22396.809,E2 -22396.809} C_VEL
LIN {X 0,Y 184.077,Z 393.669,A -85,B 0,C 180,E1 -22398.995,E2 -22398.995} C_VEL
LIN {X 0,Y 183.544,Z 395.473,A -85,B 0,C 180,E1 -22401.19,E2 -22401.19} C_VEL
LIN {X 0,Y 183.106,Z 397.933,A -85,B 0,C 180,E1 -22405.597,E2 -22405.597} C_VEL
LIN {X 0,Y 183.07,Z 398.527,A -85,B 0,C 180,E1 -22407.8,E2 -22407.8} C_VEL
LIN {X 0,Y 183.156,Z 398.686,A -85,B 0,C 180,E1 -22410,E2 -22410} C_VEL
LIN {X 0,Y 183.061,Z 398.23,A -85,B 0,C 180,E1 -22413.3,E2 -22413.3} C_VEL
LIN {X 0,Y 183.253,Z 396.868,A -85,B 0,C 180,E1 -22416.607,E2 -22416.607} C_VEL
LIN {X 0,Y 183.552,Z 395.473,A -85,B 0,C 180,E1 -22418.81,E2 -22418.81} C_VEL
LIN {X 0,Y 184.39,Z 392.516,A -85,B 0,C 180,E1 -22422.101,E2 -22422.101} C_VEL
LIN {X 0,Y 185.68,Z 388.519,A -85,B 0,C 180,E1 -22425.364,E2 -22425.364} C_VEL
LIN {X 0,Y 186.798,Z 385.689,A -85,B 0,C 180,E1 -22427.254,E2 -22427.254} C_VEL
LIN {X 0,Y 187.218,Z 383.046,A -85,B 0,C 180,E1 -22428.868,E2 -22428.868} C_VEL
LIN {X 0,Y 186.325,Z 378.214,A -85,B 0,C 180,E1 -22431.511,E2 -22431.511} C_VEL
LIN {X 0,Y 185.619,Z 372.875,A -85,B 0,C 180,E1 -22434.079,E2 -22434.079} C_VEL
LIN {X 0,Y 186.327,Z 369.244,A -85,B 0,C 180,E1 -22435.526,E2 -22435.526} C_VEL
LIN {X 0,Y 189.461,Z 360.628,A -85,B 0,C 180,E1 -22438.226,E2 -22438.226} C_VEL
LIN {X 0,Y 190.635,Z 356.784,A -85,B 0,C 180,E1 -22439.24,E2 -22439.24} C_VEL
LIN {X 0,Y 191.198,Z 349.187,A -85,B 0,C 180,E1 -22441.315,E2 -22441.315} C_VEL
LIN {X 0,Y 191.153,Z 341.763,A -85,B 0,C 180,E1 -22443.178,E2 -22443.178} C_VEL
LIN {X 0,Y 190.559,Z 333.243,A -85,B 0,C 180,E1 -22445.149,E2 -22445.149} C_VEL
LIN {X 0,Y 189.242,Z 324.064,A -85,B 0,C 180,E1 -22447.136,E2 -22447.136} C_VEL
LIN {X 0,Y 187.421,Z 315.593,A -85,B 0,C 180,E1 -22448.899,E2 -22448.899} C_VEL
LIN {X 0,Y 184.156,Z 304.904,A -85,B 0,C 180,E1 -22451.088,E2 -22451.088} C_VEL
LIN {X 0,Y 181.163,Z 297.444,A -85,B 0,C 180,E1 -22452.695,E2 -22452.695} C_VEL
LIN {X 0,Y 179.696,Z 294.366,A -85,B 0,C 180,E1 -22453.357,E2 -22453.357} C_VEL
LIN {X 0,Y 179.443,Z 293.023,A -85,B 0,C 180,E1 -22453.558,E2 -22453.558} C_VEL
LIN {X 0,Y 179.428,Z 290.746,A -85,B 0,C 180,E1 -22458.236,E2 -22458.236} C_VEL
LIN {X 0,Y 179.218,Z 289.279,A -85,B 0,C 180,E1 -22461.654,E2 -22461.654} C_VEL
LIN {X 0,Y 178.933,Z 287.302,A -85,B 0,C 180,E1 -22466.628,E2 -22466.628} C_VEL
LIN {X 0,Y 178.674,Z 285.511,A -85,B 0,C 180,E1 -22471.822,E2 -22471.822} C_VEL
LIN {X 0,Y 178.497,Z 284.002,A -85,B 0,C 180,E1 -22476.8,E2 -22476.8} C_VEL
LIN {X 0,Y 178.614,Z 283.74,A -85,B 0,C 180,E1 -22481.64,E2 -22481.64} C_VEL
LIN {X 0,Y 178.631,Z 283.735,A -85,B 0,C 180,E1 -22486.333,E2 -22486.333} C_VEL
LIN {X 0,Y 178.907,Z 283.7,A -85,B 0,C 180,E1 -22490.947,E2 -22490.947} C_VEL
LIN {X 0,Y 179.121,Z 283.671,A -85,B 0,C 180,E1 -22497.738,E2 -22497.738} C_VEL
LIN {X 0,Y 179.34,Z 283.624,A -85,B 0,C 180,E1 -22499.987,E2 -22499.987} C_VEL
LIN {X 0,Y 178.834,Z 283.691,A -85,B 0,C 180,E1 -22504.495,E2 -22504.495} C_VEL
LIN {X 0,Y 178.897,Z 283.695,A -85,B 0,C 180,E1 -22509.027,E2 -22509.027} C_VEL
LIN {X 0,Y 178.63,Z 283.73,A -85,B 0,C 180,E1 -22513.64,E2 -22513.64} C_VEL
LIN {X 0,Y 178.54,Z 283.739,A -85,B 0,C 180,E1 -22519.141,E2 -22519.141} C_VEL
LIN {X 0,Y 178.498,Z 283.742,A -85,B 0,C 180,E1 -22525.101,E2 -22525.101} C_VEL
LIN {X 0,Y 178.498,Z 283.751,A -85,B 0,C 180,E1 -22529.981,E2 -22529.981} C_VEL
LIN {X 0,Y 178.456,Z 283.755,A -85,B 0,C 180,E1 -22534.207,E2 -22534.207} C_VEL
LIN {X 0,Y 178.441,Z 283.758,A -85,B 0,C 180,E1 -22539.043,E2 -22539.043} C_VEL
LIN {X 0,Y 178.469,Z 283.755,A -85,B 0,C 180,E1 -22542.004,E2 -22542.004} C_VEL
LIN {X 0,Y 178.497,Z 283.758,A -85,B 0,C 180,E1 -22546.066,E2 -22546.066} C_VEL
LIN {X 0,Y 179.412,Z 286.482,A -85,B 0,C 180,E1 -22546.548,E2 -22546.548} C_VEL
LIN {X 0,Y 181.356,Z 289.022,A -85,B 0,C 180,E1 -22547.318,E2 -22547.318} C_VEL
LIN {X 0,Y 183.445,Z 292.456,A -85,B 0,C 180,E1 -22548.273,E2 -22548.273} C_VEL
LIN {X 0,Y 187.756,Z 300.098,A -85,B 0,C 180,E1 -22550.26,E2 -22550.26} C_VEL
LIN {X 0,Y 192.666,Z 310.537,A -85,B 0,C 180,E1 -22552.907,E2 -22552.907} C_VEL
LIN {X 0,Y 196.365,Z 320.36,A -85,B 0,C 180,E1 -22555.379,E2 -22555.379} C_VEL
LIN {X 0,Y 198.689,Z 328.104,A -85,B 0,C 180,E1 -22557.358,E2 -22557.358} C_VEL
LIN {X 0,Y 201.142,Z 337.45,A -85,B 0,C 180,E1 -22559.956,E2 -22559.956} C_VEL
LIN {X 0,Y 204.009,Z 345.211,A -85,B 0,C 180,E1 -22562.475,E2 -22562.475} C_VEL
LIN {X 0,Y 208.419,Z 353.198,A -85,B 0,C 180,E1 -22565.533,E2 -22565.533} C_VEL
LIN {X 0,Y 213.094,Z 359.483,A -85,B 0,C 180,E1 -22568.273,E2 -22568.273} C_VEL
LIN {X 0,Y 219.189,Z 365.566,A -85,B 0,C 180,E1 -22571.299,E2 -22571.299} C_VEL
LIN {X 0,Y 226.22,Z 370.909,A -85,B 0,C 180,E1 -22574.332,E2 -22574.332} C_VEL
LIN {X 0,Y 233.47,Z 375.262,A -85,B 0,C 180,E1 -22577.155,E2 -22577.155} C_VEL
LIN {X 0,Y 242.322,Z 379.419,A -85,B 0,C 180,E1 -22580.354,E2 -22580.354} C_VEL
LIN {X 0,Y 248.075,Z 381.668,A -85,B 0,C 180,E1 -22582.45,E2 -22582.45} C_VEL
LIN {X 0,Y 253.989,Z 383.646,A -85,B 0,C 180,E1 -22584.82,E2 -22584.82} C_VEL
LIN {X 0,Y 254.967,Z 383.933,A -85,B 0,C 180,E1 -22585.257,E2 -22585.257} C_VEL
LIN {X 0,Y 257.746,Z 384.858,A -85,B 0,C 180,E1 -22586.874,E2 -22586.874} C_VEL
LIN {X 0,Y 260.163,Z 385.366,A -85,B 0,C 180,E1 -22588.452,E2 -22588.452} C_VEL
LIN {X 0,Y 261.74,Z 385.505,A -85,B 0,C 180,E1 -22590,E2 -22590} C_VEL
LIN {X 0,Y 260.079,Z 385.355,A -85,B 0,C 180,E1 -22591.588,E2 -22591.588} C_VEL
LIN {X 0,Y 257.736,Z 384.858,A -85,B 0,C 180,E1 -22593.126,E2 -22593.126} C_VEL
LIN {X 0,Y 254.966,Z 383.933,A -85,B 0,C 180,E1 -22594.743,E2 -22594.743} C_VEL
LIN {X 0,Y 250.886,Z 382.691,A -85,B 0,C 180,E1 -22596.433,E2 -22596.433} C_VEL
LIN {X 0,Y 246.321,Z 381.032,A -85,B 0,C 180,E1 -22598.202,E2 -22598.202} C_VEL
LIN {X 0,Y 241.157,Z 378.923,A -85,B 0,C 180,E1 -22600.07,E2 -22600.07} C_VEL
LIN {X 0,Y 231.371,Z 374.127,A -85,B 0,C 180,E1 -22603.644,E2 -22603.644} C_VEL
LIN {X 0,Y 223.656,Z 369.124,A -85,B 0,C 180,E1 -22606.747,E2 -22606.747} C_VEL
LIN {X 0,Y 216.7,Z 363.271,A -85,B 0,C 180,E1 -22609.902,E2 -22609.902} C_VEL
LIN {X 0,Y 210.384,Z 356.122,A -85,B 0,C 180,E1 -22613.247,E2 -22613.247} C_VEL
LIN {X 0,Y 205.58,Z 348.294,A -85,B 0,C 180,E1 -22616.386,E2 -22616.386} C_VEL
LIN {X 0,Y 202.516,Z 341.254,A -85,B 0,C 180,E1 -22618.838,E2 -22618.838} C_VEL
LIN {X 0,Y 200.082,Z 333.676,A -85,B 0,C 180,E1 -22621.139,E2 -22621.139} C_VEL
LIN {X 0,Y 197.738,Z 324.749,A -85,B 0,C 180,E1 -22623.503,E2 -22623.503} C_VEL
LIN {X 0,Y 194.344,Z 314.862,A -85,B 0,C 180,E1 -22626.012,E2 -22626.012} C_VEL
LIN {X 0,Y 190.837,Z 306.523,A -85,B 0,C 180,E1 -22628.11,E2 -22628.11} C_VEL
LIN {X 0,Y 185.684,Z 296.27,A -85,B 0,C 180,E1 -22630.71,E2 -22630.71} C_VEL
LIN {X 0,Y 181.353,Z 289.041,A -85,B 0,C 180,E1 -22632.681,E2 -22632.681} C_VEL
LIN {X 0,Y 179.951,Z 287.248,A -85,B 0,C 180,E1 -22633.248,E2 -22633.248} C_VEL
LIN {X 0,Y 178.675,Z 284.649,A -85,B 0,C 180,E1 -22633.841,E2 -22633.841} C_VEL
LIN {X 0,Y 178.496,Z 283.751,A -85,B 0,C 180,E1 -22633.985,E2 -22633.985} C_VEL
LIN {X 0,Y 178.47,Z 283.754,A -85,B 0,C 180,E1 -22638.434,E2 -22638.434} C_VEL
LIN {X 0,Y 178.429,Z 283.758,A -85,B 0,C 180,E1 -22643.803,E2 -22643.803} C_VEL
LIN {X 0,Y 178.463,Z 283.753,A -85,B 0,C 180,E1 -22646.56,E2 -22646.56} C_VEL
LIN {X 0,Y 178.498,Z 283.751,A -85,B 0,C 180,E1 -22650.019,E2 -22650.019} C_VEL
LIN {X 0,Y 178.498,Z 283.742,A -85,B 0,C 180,E1 -22654.899,E2 -22654.899} C_VEL
LIN {X 0,Y 178.54,Z 283.739,A -85,B 0,C 180,E1 -22660.859,E2 -22660.859} C_VEL
LIN {X 0,Y 178.63,Z 283.73,A -85,B 0,C 180,E1 -22666.36,E2 -22666.36} C_VEL
LIN {X 0,Y 178.897,Z 283.695,A -85,B 0,C 180,E1 -22670.973,E2 -22670.973} C_VEL
LIN {X 0,Y 178.834,Z 283.691,A -85,B 0,C 180,E1 -22675.505,E2 -22675.505} C_VEL
LIN {X 0,Y 179.34,Z 283.624,A -85,B 0,C 180,E1 -22680.013,E2 -22680.013} C_VEL
LIN {X 0,Y 178.831,Z 283.709,A -85,B 0,C 180,E1 -22684.521,E2 -22684.521} C_VEL
LIN {X 0,Y 178.907,Z 283.7,A -85,B 0,C 180,E1 -22689.053,E2 -22689.053} C_VEL
LIN {X 0,Y 178.631,Z 283.737,A -85,B 0,C 180,E1 -22693.667,E2 -22693.667} C_VEL
LIN {X 0,Y 178.562,Z 283.743,A -85,B 0,C 180,E1 -22699.162,E2 -22699.162} C_VEL
LIN {X 0,Y 178.505,Z 283.992,A -85,B 0,C 180,E1 -22703.199,E2 -22703.199} C_VEL
LIN {X 0,Y 178.616,Z 284.709,A -85,B 0,C 180,E1 -22705.659,E2 -22705.659} C_VEL
LIN {X 0,Y 178.779,Z 286.365,A -85,B 0,C 180,E1 -22710.747,E2 -22710.747} C_VEL
LIN {X 0,Y 179.007,Z 287.723,A -85,B 0,C 180,E1 -22714.465,E2 -22714.465} C_VEL
LIN {X 0,Y 179.253,Z 289.498,A -85,B 0,C 180,E1 -22718.866,E2 -22718.866} C_VEL
LIN {X 0,Y 179.43,Z 290.822,A -85,B 0,C 180,E1 -22721.911,E2 -22721.911} C_VEL
LIN {X 0,Y 179.449,Z 293.039,A -85,B 0,C 180,E1 -22726.446,E2 -22726.446} C_VEL
LIN {X 0,Y 180.409,Z 296.19,A -85,B 0,C 180,E1 -22726.984,E2 -22726.984} C_VEL
LIN {X 0,Y 181.745,Z 298.714,A -85,B 0,C 180,E1 -22727.6,E2 -22727.6} C_VEL
LIN {X 0,Y 184.746,Z 306.494,A -85,B 0,C 180,E1 -22729.232,E2 -22729.232} C_VEL
LIN {X 0,Y 188.14,Z 318.487,A -85,B 0,C 180,E1 -22731.686,E2 -22731.686} C_VEL
LIN {X 0,Y 190.112,Z 329.547,A -85,B 0,C 180,E1 -22734.029,E2 -22734.029} C_VEL
LIN {X 0,Y 191.017,Z 339.083,A -85,B 0,C 180,E1 -22736.176,E2 -22736.176} C_VEL
LIN {X 0,Y 191.229,Z 347.908,A -85,B 0,C 180,E1 -22738.346,E2 -22738.346} C_VEL
LIN {X 0,Y 190.913,Z 354.851,A -85,B 0,C 180,E1 -22740.201,E2 -22740.201} C_VEL
LIN {X 0,Y 190.152,Z 358.71,A -85,B 0,C 180,E1 -22741.284,E2 -22741.284} C_VEL
LIN {X 0,Y 187.041,Z 367.262,A -85,B 0,C 180,E1 -22743.801,E2 -22743.801} C_VEL
LIN {X 0,Y 184.201,Z 375.307,A -85,B 0,C 180,E1 -22746.83,E2 -22746.83} C_VEL
LIN {X 0,Y 181.736,Z 381.259,A -85,B 0,C 180,E1 -22749.633,E2 -22749.633} C_VEL
LIN {X 0,Y 179.471,Z 386.752,A -85,B 0,C 180,E1 -22752.921,E2 -22752.921} C_VEL
LIN {X 0,Y 177.842,Z 391.084,A -85,B 0,C 180,E1 -22756.284,E2 -22756.284} C_VEL
LIN {X 0,Y 177.074,Z 393.456,A -85,B 0,C 180,E1 -22758.554,E2 -22758.554} C_VEL
LIN {X 0,Y 176.507,Z 395.261,A -85,B 0,C 180,E1 -22760.836,E2 -22760.836} C_VEL
LIN {X 0,Y 176.037,Z 397.722,A -85,B 0,C 180,E1 -22765.42,E2 -22765.42} C_VEL
LIN {X 0,Y 175.979,Z 398.316,A -85,B 0,C 180,E1 -22767.711,E2 -22767.711} C_VEL
LIN {X 0,Y 176.065,Z 398.475,A -85,B 0,C 180,E1 -22770,E2 -22770} C_VEL
LIN {X 0,Y 175.977,Z 398.122,A -85,B 0,C 180,E1 -22773.036,E2 -22773.036} C_VEL
LIN {X 0,Y 176.037,Z 397.722,A -85,B 0,C 180,E1 -22774.58,E2 -22774.58} C_VEL
LIN {X 0,Y 176.513,Z 395.261,A -85,B 0,C 180,E1 -22779.164,E2 -22779.164} C_VEL
LIN {X 0,Y 177.44,Z 392.304,A -85,B 0,C 180,E1 -22782.582,E2 -22782.582} C_VEL
LIN {X 0,Y 178.809,Z 388.306,A -85,B 0,C 180,E1 -22785.97,E2 -22785.97} C_VEL
LIN {X 0,Y 180.94,Z 383.176,A -85,B 0,C 180,E1 -22789.278,E2 -22789.278} C_VEL
LIN {X 0,Y 183.058,Z 377.911,A -85,B 0,C 180,E1 -22791.982,E2 -22791.982} C_VEL
LIN {X 0,Y 185.214,Z 372.265,A -85,B 0,C 180,E1 -22794.377,E2 -22794.377} C_VEL
LIN {X 0,Y 186.327,Z 369.244,A -85,B 0,C 180,E1 -22795.526,E2 -22795.526} C_VEL
LIN {X 0,Y 187.04,Z 365.518,A -85,B 0,C 180,E1 -22796.922,E2 -22796.922} C_VEL
LIN {X 0,Y 186.784,Z 361.707,A -85,B 0,C 180,E1 -22798.326,E2 -22798.326} C_VEL
LIN {X 0,Y 185.195,Z 353.823,A -85,B 0,C 180,E1 -22801.084,E2 -22801.084} C_VEL
LIN {X 0,Y 184.792,Z 347.945,A -85,B 0,C 180,E1 -22802.818,E2 -22802.818} C_VEL
LIN {X 0,Y 184.633,Z 339.164,A -85,B 0,C 180,E1 -22805.086,E2 -22805.086} C_VEL
LIN {X 0,Y 183.692,Z 329.332,A -85,B 0,C 180,E1 -22807.433,E2 -22807.433} C_VEL
LIN {X 0,Y 181.957,Z 319.482,A -85,B 0,C 180,E1 -22809.651,E2 -22809.651} C_VEL
LIN {X 0,Y 178.908,Z 308.409,A -85,B 0,C 180,E1 -22812.128,E2 -22812.128} C_VEL
LIN {X 0,Y 176.188,Z 301.535,A -85,B 0,C 180,E1 -22813.73,E2 -22813.73} C_VEL
LIN {X 0,Y 174.457,Z 297.521,A -85,B 0,C 180,E1 -22814.726,E2 -22814.726} C_VEL
LIN {X 0,Y 172.709,Z 294.261,A -85,B 0,C 180,E1 -22815.573,E2 -22815.573} C_VEL
LIN {X 0,Y 172.388,Z 292.727,A -85,B 0,C 180,E1 -22815.855,E2 -22815.855} C_VEL
LIN {X 0,Y 172.221,Z 290.565,A -85,B 0,C 180,E1 -22820.836,E2 -22820.836} C_VEL
LIN {X 0,Y 171.993,Z 288.9,A -85,B 0,C 180,E1 -22825.091,E2 -22825.091} C_VEL
LIN {X 0,Y 171.687,Z 286.969,A -85,B 0,C 180,E1 -22830.566,E2 -22830.566} C_VEL
LIN {X 0,Y 171.503,Z 285.398,A -85,B 0,C 180,E1 -22835.795,E2 -22835.795} C_VEL
LIN {X 0,Y 171.432,Z 284.717,A -85,B 0,C 180,E1 -22838.335,E2 -22838.335} C_VEL
LIN {X 0,Y 171.515,Z 284.624,A -85,B 0,C 180,E1 -22840.851,E2 -22840.851} C_VEL
LIN {X 0,Y 171.547,Z 284.617,A -85,B 0,C 180,E1 -22845.757,E2 -22845.757} C_VEL
LIN {X 0,Y 171.846,Z 284.58,A -85,B 0,C 180,E1 -22850.572,E2 -22850.572} C_VEL
LIN {X 0,Y 171.781,Z 284.588,A -85,B 0,C 180,E1 -22855.293,E2 -22855.293} C_VEL
LIN {X 0,Y 172.305,Z 284.499,A -85,B 0,C 180,E1 -22859.986,E2 -22859.986} C_VEL
LIN {X 0,Y 171.784,Z 284.571,A -85,B 0,C 180,E1 -22864.679,E2 -22864.679} C_VEL
LIN {X 0,Y 171.835,Z 284.573,A -85,B 0,C 180,E1 -22869.401,E2 -22869.401} C_VEL
LIN {X 0,Y 171.544,Z 284.61,A -85,B 0,C 180,E1 -22874.215,E2 -22874.215} C_VEL
LIN {X 0,Y 171.467,Z 284.618,A -85,B 0,C 180,E1 -22879.491,E2 -22879.491} C_VEL
LIN {X 0,Y 171.437,Z 284.623,A -85,B 0,C 180,E1 -22885.596,E2 -22885.596} C_VEL
LIN {X 0,Y 171.416,Z 284.633,A -85,B 0,C 180,E1 -22890.574,E2 -22890.574} C_VEL
LIN {X 0,Y 171.375,Z 284.638,A -85,B 0,C 180,E1 -22895.02,E2 -22895.02} C_VEL
LIN {X 0,Y 171.395,Z 284.635,A -85,B 0,C 180,E1 -22898.824,E2 -22898.824} C_VEL
LIN {X 0,Y 171.413,Z 284.829,A -85,B 0,C 180,E1 -22903.8,E2 -22903.8} C_VEL
LIN {X 0,Y 172.454,Z 287.539,A -85,B 0,C 180,E1 -22904.377,E2 -22904.377} C_VEL
LIN {X 0,Y 174.471,Z 289.895,A -85,B 0,C 180,E1 -22905.253,E2 -22905.253} C_VEL
LIN {X 0,Y 176.338,Z 293.172,A -85,B 0,C 180,E1 -22906.228,E2 -22906.228} C_VEL
LIN {X 0,Y 180.852,Z 300.821,A -85,B 0,C 180,E1 -22908.483,E2 -22908.483} C_VEL
LIN {X 0,Y 186.114,Z 311.874,A -85,B 0,C 180,E1 -22911.556,E2 -22911.556} C_VEL
LIN {X 0,Y 189.303,Z 320.291,A -85,B 0,C 180,E1 -22913.825,E2 -22913.825} C_VEL
LIN {X 0,Y 192.01,Z 328.962,A -85,B 0,C 180,E1 -22916.221,E2 -22916.221} C_VEL
LIN {X 0,Y 194.087,Z 337.78,A -85,B 0,C 180,E1 -22918.769,E2 -22918.769} C_VEL
LIN {X 0,Y 196.866,Z 346.479,A -85,B 0,C 180,E1 -22921.705,E2 -22921.705} C_VEL
LIN {X 0,Y 200.427,Z 353.665,A -85,B 0,C 180,E1 -22924.563,E2 -22924.563} C_VEL
LIN {X 0,Y 205.097,Z 360.446,A -85,B 0,C 180,E1 -22927.66,E2 -22927.66} C_VEL
LIN {X 0,Y 210.187,Z 365.843,A -85,B 0,C 180,E1 -22930.466,E2 -22930.466} C_VEL
LIN {X 0,Y 216.565,Z 370.966,A -85,B 0,C 180,E1 -22933.492,E2 -22933.492} C_VEL
LIN {X 0,Y 223.927,Z 375.521,A -85,B 0,C 180,E1 -22936.581,E2 -22936.581} C_VEL
LIN {X 0,Y 231.681,Z 379.204,A -85,B 0,C 180,E1 -22939.513,E2 -22939.513} C_VEL
LIN {X 0,Y 237.123,Z 381.309,A -85,B 0,C 180,E1 -22941.478,E2 -22941.478} C_VEL
LIN {X 0,Y 242.196,Z 382.953,A -85,B 0,C 180,E1 -22943.335,E2 -22943.335} C_VEL
LIN {X 0,Y 246.792,Z 384.24,A -85,B 0,C 180,E1 -22945.192,E2 -22945.192} C_VEL
LIN {X 0,Y 249.977,Z 385.091,A -85,B 0,C 180,E1 -22946.777,E2 -22946.777} C_VEL
LIN {X 0,Y 253.02,Z 385.654,A -85,B 0,C 180,E1 -22948.669,E2 -22948.669} C_VEL
LIN {X 0,Y 254.437,Z 385.718,A -85,B 0,C 180,E1 -22950,E2 -22950} C_VEL
LIN {X 0,Y 252.571,Z 385.591,A -85,B 0,C 180,E1 -22951.594,E2 -22951.594} C_VEL
LIN {X 0,Y 249.971,Z 385.091,A -85,B 0,C 180,E1 -22953.223,E2 -22953.223} C_VEL
LIN {X 0,Y 246.548,Z 384.181,A -85,B 0,C 180,E1 -22954.906,E2 -22954.906} C_VEL
LIN {X 0,Y 240.792,Z 382.495,A -85,B 0,C 180,E1 -22957.195,E2 -22957.195} C_VEL
LIN {X 0,Y 234.969,Z 380.486,A -85,B 0,C 180,E1 -22959.317,E2 -22959.317} C_VEL
LIN {X 0,Y 226.156,Z 376.653,A -85,B 0,C 180,E1 -22962.564,E2 -22962.564} C_VEL
LIN {X 0,Y 218.792,Z 372.443,A -85,B 0,C 180,E1 -22965.547,E2 -22965.547} C_VEL
LIN {X 0,Y 211.578,Z 367.056,A -85,B 0,C 180,E1 -22968.841,E2 -22968.841} C_VEL
LIN {X 0,Y 205.499,Z 360.933,A -85,B 0,C 180,E1 -22972.098,E2 -22972.098} C_VEL
LIN {X 0,Y 201.271,Z 355.086,A -85,B 0,C 180,E1 -22974.822,E2 -22974.822} C_VEL
LIN {X 0,Y 197.417,Z 347.618,A -85,B 0,C 180,E1 -22977.854,E2 -22977.854} C_VEL
LIN {X 0,Y 194.912,Z 340.601,A -85,B 0,C 180,E1 -22980.318,E2 -22980.318} C_VEL
LIN {X 0,Y 193.021,Z 333.291,A -85,B 0,C 180,E1 -22982.559,E2 -22982.559} C_VEL
LIN {X 0,Y 191.287,Z 326.255,A -85,B 0,C 180,E1 -22984.537,E2 -22984.537} C_VEL
LIN {X 0,Y 187.907,Z 316.442,A -85,B 0,C 180,E1 -22987.224,E2 -22987.224} C_VEL
LIN {X 0,Y 184.305,Z 307.829,A -85,B 0,C 180,E1 -22989.574,E2 -22989.574} C_VEL
LIN {X 0,Y 178.811,Z 297.291,A -85,B 0,C 180,E1 -22992.551,E2 -22992.551} C_VEL
LIN {X 0,Y 175.952,Z 292.677,A -85,B 0,C 180,E1 -22993.951,E2 -22993.951} C_VEL
LIN {X 0,Y 173.974,Z 289.196,A -85,B 0,C 180,E1 -22994.978,E2 -22994.978} C_VEL
LIN {X 0,Y 172.14,Z 286.968,A -85,B 0,C 180,E1 -22995.796,E2 -22995.796} C_VEL
LIN {X 0,Y 171.401,Z 284.635,A -85,B 0,C 180,E1 -22996.318,E2 -22996.318} C_VEL
LIN {X 0,Y 171.406,Z 284.633,A -85,B 0,C 180,E1 -23002.066,E2 -23002.066} C_VEL
LIN {X 0,Y 171.393,Z 284.636,A -85,B 0,C 180,E1 -23007.805,E2 -23007.805} C_VEL
LIN {X 0,Y 171.424,Z 284.632,A -85,B 0,C 180,E1 -23010.547,E2 -23010.547} C_VEL
LIN {X 0,Y 171.422,Z 284.626,A -85,B 0,C 180,E1 -23015.813,E2 -23015.813} C_VEL
LIN {X 0,Y 171.494,Z 284.616,A -85,B 0,C 180,E1 -23020.877,E2 -23020.877} C_VEL
LIN {X 0,Y 171.544,Z 284.61,A -85,B 0,C 180,E1 -23025.785,E2 -23025.785} C_VEL
LIN {X 0,Y 171.835,Z 284.573,A -85,B 0,C 180,E1 -23030.599,E2 -23030.599} C_VEL
LIN {X 0,Y 171.784,Z 284.571,A -85,B 0,C 180,E1 -23035.321,E2 -23035.321} C_VEL
LIN {X 0,Y 172.305,Z 284.499,A -85,B 0,C 180,E1 -23040.014,E2 -23040.014} C_VEL
LIN {X 0,Y 171.781,Z 284.587,A -85,B 0,C 180,E1 -23044.707,E2 -23044.707} C_VEL
LIN {X 0,Y 171.846,Z 284.58,A -85,B 0,C 180,E1 -23049.428,E2 -23049.428} C_VEL
LIN {X 0,Y 171.547,Z 284.618,A -85,B 0,C 180,E1 -23054.243,E2 -23054.243} C_VEL
LIN {X 0,Y 171.486,Z 284.624,A -85,B 0,C 180,E1 -23059.509,E2 -23059.509} C_VEL
LIN {X 0,Y 171.434,Z 284.711,A -85,B 0,C 180,E1 -23061.665,E2 -23061.665} C_VEL
LIN {X 0,Y 171.591,Z 286.141,A -85,B 0,C 180,E1 -23066.792,E2 -23066.792} C_VEL
LIN {X 0,Y 171.814,Z 287.905,A -85,B 0,C 180,E1 -23072.138,E2 -23072.138} C_VEL
LIN {X 0,Y 172.002,Z 289.015,A -85,B 0,C 180,E1 -23075.196,E2 -23075.196} C_VEL
LIN {X 0,Y 172.222,Z 290.567,A -85,B 0,C 180,E1 -23079.165,E2 -23079.165} C_VEL
LIN {X 0,Y 172.403,Z 292.808,A -85,B 0,C 180,E1 -23084.205,E2 -23084.205} C_VEL
LIN {X 0,Y 173.487,Z 296.017,A -85,B 0,C 180,E1 -23084.821,E2 -23084.821} C_VEL
LIN {X 0,Y 174.983,Z 298.544,A -85,B 0,C 180,E1 -23085.556,E2 -23085.556} C_VEL
LIN {X 0,Y 178.516,Z 307.169,A -85,B 0,C 180,E1 -23087.591,E2 -23087.591} C_VEL
LIN {X 0,Y 181.948,Z 319.435,A -85,B 0,C 180,E1 -23090.338,E2 -23090.338} C_VEL
LIN {X 0,Y 183.718,Z 329.253,A -85,B 0,C 180,E1 -23092.556,E2 -23092.556} C_VEL
LIN {X 0,Y 184.614,Z 338.026,A -85,B 0,C 180,E1 -23094.632,E2 -23094.632} C_VEL
LIN {X 0,Y 184.787,Z 347.681,A -85,B 0,C 180,E1 -23097.106,E2 -23097.106} C_VEL
LIN {X 0,Y 184.469,Z 354.629,A -85,B 0,C 180,E1 -23099.048,E2 -23099.048} C_VEL
LIN {X 0,Y 183.865,Z 358.495,A -85,B 0,C 180,E1 -23100.205,E2 -23100.205} C_VEL
LIN {X 0,Y 180.679,Z 367.05,A -85,B 0,C 180,E1 -23102.804,E2 -23102.804} C_VEL
LIN {X 0,Y 177.54,Z 375.364,A -85,B 0,C 180,E1 -23106.049,E2 -23106.049} C_VEL
LIN {X 0,Y 175.044,Z 381.046,A -85,B 0,C 180,E1 -23108.817,E2 -23108.817} C_VEL
LIN {X 0,Y 172.677,Z 386.54,A -85,B 0,C 180,E1 -23112.227,E2 -23112.227} C_VEL
LIN {X 0,Y 170.924,Z 390.872,A -85,B 0,C 180,E1 -23115.718,E2 -23115.718} C_VEL
LIN {X 0,Y 170.098,Z 393.244,A -85,B 0,C 180,E1 -23118.078,E2 -23118.078} C_VEL
LIN {X 0,Y 169.489,Z 395.049,A -85,B 0,C 180,E1 -23120.453,E2 -23120.453} C_VEL
LIN {X 0,Y 168.96,Z 397.51,A -85,B 0,C 180,E1 -23125.228,E2 -23125.228} C_VEL
LIN {X 0,Y 168.889,Z 398.104,A -85,B 0,C 180,E1 -23127.615,E2 -23127.615} C_VEL
LIN {X 0,Y 168.977,Z 398.264,A -85,B 0,C 180,E1 -23130,E2 -23130} C_VEL
LIN {X 0,Y 168.88,Z 398.044,A -85,B 0,C 180,E1 -23132.626,E2 -23132.626} C_VEL
LIN {X 0,Y 168.96,Z 397.51,A -85,B 0,C 180,E1 -23134.772,E2 -23134.772} C_VEL
LIN {X 0,Y 169.494,Z 395.05,A -85,B 0,C 180,E1 -23139.547,E2 -23139.547} C_VEL
LIN {X 0,Y 170.484,Z 392.092,A -85,B 0,C 180,E1 -23143.104,E2 -23143.104} C_VEL
LIN {X 0,Y 171.966,Z 388.094,A -85,B 0,C 180,E1 -23146.623,E2 -23146.623} C_VEL
LIN {X 0,Y 174.23,Z 382.963,A -85,B 0,C 180,E1 -23150.051,E2 -23150.051} C_VEL
LIN {X 0,Y 176.489,Z 377.7,A -85,B 0,C 180,E1 -23152.846,E2 -23152.846} C_VEL
LIN {X 0,Y 178.982,Z 371.377,A -85,B 0,C 180,E1 -23155.59,E2 -23155.59} C_VEL
LIN {X 0,Y 181.276,Z 365.422,A -85,B 0,C 180,E1 -23157.725,E2 -23157.725} C_VEL
LIN {X 0,Y 183.833,Z 358.494,A -85,B 0,C 180,E1 -23159.801,E2 -23159.801} C_VEL
LIN {X 0,Y 184.668,Z 351.392,A -85,B 0,C 180,E1 -23161.873,E2 -23161.873} C_VEL
LIN {X 0,Y 184.792,Z 347.945,A -85,B 0,C 180,E1 -23162.818,E2 -23162.818} C_VEL
LIN {X 0,Y 184.324,Z 343.708,A -85,B 0,C 180,E1 -23164.084,E2 -23164.084} C_VEL
LIN {X 0,Y 182.863,Z 339.811,A -85,B 0,C 180,E1 -23165.412,E2 -23165.412} C_VEL
LIN {X 0,Y 178.922,Z 332.152,A -85,B 0,C 180,E1 -23168.079,E2 -23168.079} C_VEL
LIN {X 0,Y 177.355,Z 327.834,A -85,B 0,C 180,E1 -23169.326,E2 -23169.326} C_VEL
LIN {X 0,Y 177.007,Z 326.259,A -85,B 0,C 180,E1 -23169.71,E2 -23169.71} C_VEL
LIN {X 0,Y 174.599,Z 315.333,A -85,B 0,C 180,E1 -23172.345,E2 -23172.345} C_VEL
LIN {X 0,Y 171.745,Z 306.469,A -85,B 0,C 180,E1 -23174.562,E2 -23174.562} C_VEL
LIN {X 0,Y 169.67,Z 301.891,A -85,B 0,C 180,E1 -23175.798,E2 -23175.798} C_VEL
LIN {X 0,Y 167.661,Z 297.554,A -85,B 0,C 180,E1 -23177.037,E2 -23177.037} C_VEL
LIN {X 0,Y 165.851,Z 294.717,A -85,B 0,C 180,E1 -23177.981,E2 -23177.981} C_VEL
LIN {X 0,Y 165.257,Z 292.42,A -85,B 0,C 180,E1 -23178.478,E2 -23178.478} C_VEL
LIN {X 0,Y 165.004,Z 290.522,A -85,B 0,C 180,E1 -23183.38,E2 -23183.38} C_VEL
LIN {X 0,Y 164.75,Z 288.498,A -85,B 0,C 180,E1 -23189.195,E2 -23189.195} C_VEL
LIN {X 0,Y 164.548,Z 286.799,A -85,B 0,C 180,E1 -23194.702,E2 -23194.702} C_VEL
LIN {X 0,Y 164.426,Z 285.508,A -85,B 0,C 180,E1 -23200.106,E2 -23200.106} C_VEL
LIN {X 0,Y 164.477,Z 285.498,A -85,B 0,C 180,E1 -23205.131,E2 -23205.131} C_VEL
LIN {X 0,Y 164.768,Z 285.462,A -85,B 0,C 180,E1 -23210.163,E2 -23210.163} C_VEL
LIN {X 0,Y 164.821,Z 285.454,A -85,B 0,C 180,E1 -23212.637,E2 -23212.637} C_VEL
LIN {X 0,Y 165.27,Z 285.373,A -85,B 0,C 180,E1 -23219.986,E2 -23219.986} C_VEL
LIN {X 0,Y 164.815,Z 285.456,A -85,B 0,C 180,E1 -23227.335,E2 -23227.335} C_VEL
LIN {X 0,Y 164.691,Z 285.466,A -85,B 0,C 180,E1 -23231.044,E2 -23231.044} C_VEL
LIN {X 0,Y 164.425,Z 285.505,A -85,B 0,C 180,E1 -23237.394,E2 -23237.394} C_VEL
LIN {X 0,Y 164.339,Z 285.515,A -85,B 0,C 180,E1 -23242.62,E2 -23242.62} C_VEL
LIN {X 0,Y 164.364,Z 285.506,A -85,B 0,C 180,E1 -23246.114,E2 -23246.114} C_VEL
LIN {X 0,Y 164.35,Z 285.511,A -85,B 0,C 180,E1 -23251.215,E2 -23251.215} C_VEL
LIN {X 0,Y 164.318,Z 285.517,A -85,B 0,C 180,E1 -23256.763,E2 -23256.763} C_VEL
LIN {X 0,Y 164.341,Z 285.514,A -85,B 0,C 180,E1 -23261.19,E2 -23261.19} C_VEL
LIN {X 0,Y 165.295,Z 288.247,A -85,B 0,C 180,E1 -23261.814,E2 -23261.814} C_VEL
LIN {X 0,Y 167.594,Z 291.025,A -85,B 0,C 180,E1 -23262.972,E2 -23262.972} C_VEL
LIN {X 0,Y 169.575,Z 294.331,A -85,B 0,C 180,E1 -23264.105,E2 -23264.105} C_VEL
LIN {X 0,Y 174.255,Z 302.257,A -85,B 0,C 180,E1 -23266.715,E2 -23266.715} C_VEL
LIN {X 0,Y 178.526,Z 310.884,A -85,B 0,C 180,E1 -23269.357,E2 -23269.357} C_VEL
LIN {X 0,Y 182.345,Z 320.365,A -85,B 0,C 180,E1 -23272.169,E2 -23272.169} C_VEL
LIN {X 0,Y 185.338,Z 329.825,A -85,B 0,C 180,E1 -23274.987,E2 -23274.987} C_VEL
LIN {X 0,Y 187.264,Z 338.294,A -85,B 0,C 180,E1 -23277.575,E2 -23277.575} C_VEL
LIN {X 0,Y 189.423,Z 346.419,A -85,B 0,C 180,E1 -23280.387,E2 -23280.387} C_VEL
LIN {X 0,Y 191.691,Z 352.377,A -85,B 0,C 180,E1 -23282.735,E2 -23282.735} C_VEL
LIN {X 0,Y 196.239,Z 360.064,A -85,B 0,C 180,E1 -23286.319,E2 -23286.319} C_VEL
LIN {X 0,Y 201.337,Z 366.117,A -85,B 0,C 180,E1 -23289.57,E2 -23289.57} C_VEL
LIN {X 0,Y 206.494,Z 370.626,A -85,B 0,C 180,E1 -23292.311,E2 -23292.311} C_VEL
LIN {X 0,Y 213.888,Z 375.471,A -85,B 0,C 180,E1 -23295.713,E2 -23295.713} C_VEL
LIN {X 0,Y 222.197,Z 379.486,A -85,B 0,C 180,E1 -23299.06,E2 -23299.06} C_VEL
LIN {X 0,Y 227.752,Z 381.592,A -85,B 0,C 180,E1 -23301.125,E2 -23301.125} C_VEL
LIN {X 0,Y 233.503,Z 383.332,A -85,B 0,C 180,E1 -23303.217,E2 -23303.217} C_VEL
LIN {X 0,Y 239.606,Z 384.823,A -85,B 0,C 180,E1 -23305.589,E2 -23305.589} C_VEL
LIN {X 0,Y 241.92,Z 385.333,A -85,B 0,C 180,E1 -23306.669,E2 -23306.669} C_VEL
LIN {X 0,Y 245.963,Z 385.908,A -85,B 0,C 180,E1 -23308.985,E2 -23308.985} C_VEL
LIN {X 0,Y 247.117,Z 385.932,A -85,B 0,C 180,E1 -23310,E2 -23310} C_VEL
LIN {X 0,Y 245.963,Z 385.908,A -85,B 0,C 180,E1 -23311.016,E2 -23311.016} C_VEL
LIN {X 0,Y 241.917,Z 385.332,A -85,B 0,C 180,E1 -23313.331,E2 -23313.331} C_VEL
LIN {X 0,Y 237.921,Z 384.435,A -85,B 0,C 180,E1 -23315.084,E2 -23315.084} C_VEL
LIN {X 0,Y 233.131,Z 383.225,A -85,B 0,C 180,E1 -23316.926,E2 -23316.926} C_VEL
LIN {X 0,Y 225.03,Z 380.59,A -85,B 0,C 180,E1 -23319.89,E2 -23319.89} C_VEL
LIN {X 0,Y 216.492,Z 376.865,A -85,B 0,C 180,E1 -23323.184,E2 -23323.184} C_VEL
LIN {X 0,Y 208.845,Z 372.328,A -85,B 0,C 180,E1 -23326.531,E2 -23326.531} C_VEL
LIN {X 0,Y 201.964,Z 366.73,A -85,B 0,C 180,E1 -23330.067,E2 -23330.067} C_VEL
LIN {X 0,Y 197.004,Z 361.2,A -85,B 0,C 180,E1 -23333.105,E2 -23333.105} C_VEL
LIN {X 0,Y 193.386,Z 355.484,A -85,B 0,C 180,E1 -23335.855,E2 -23335.855} C_VEL
LIN {X 0,Y 190.283,Z 348.792,A -85,B 0,C 180,E1 -23338.695,E2 -23338.695} C_VEL
LIN {X 0,Y 188.046,Z 341.666,A -85,B 0,C 180,E1 -23341.314,E2 -23341.314} C_VEL
LIN {X 0,Y 186.216,Z 333.559,A -85,B 0,C 180,E1 -23343.898,E2 -23343.898} C_VEL
LIN {X 0,Y 184.342,Z 326.501,A -85,B 0,C 180,E1 -23346.036,E2 -23346.036} C_VEL
LIN {X 0,Y 180.834,Z 316.341,A -85,B 0,C 180,E1 -23349.012,E2 -23349.012} C_VEL
LIN {X 0,Y 176.718,Z 307,A -85,B 0,C 180,E1 -23351.807,E2 -23351.807} C_VEL
LIN {X 0,Y 171.505,Z 297.592,A -85,B 0,C 180,E1 -23354.834,E2 -23354.834} C_VEL
LIN {X 0,Y 169.713,Z 294.463,A -85,B 0,C 180,E1 -23355.83,E2 -23355.83} C_VEL
LIN {X 0,Y 167.783,Z 291.506,A -85,B 0,C 180,E1 -23356.897,E2 -23356.897} C_VEL
LIN {X 0,Y 167.043,Z 290.225,A -85,B 0,C 180,E1 -23357.33,E2 -23357.33} C_VEL
LIN {X 0,Y 165.077,Z 287.855,A -85,B 0,C 180,E1 -23358.323,E2 -23358.323} C_VEL
LIN {X 0,Y 164.343,Z 285.513,A -85,B 0,C 180,E1 -23358.912,E2 -23358.912} C_VEL
LIN {X 0,Y 164.316,Z 285.516,A -85,B 0,C 180,E1 -23364.355,E2 -23364.355} C_VEL
LIN {X 0,Y 164.365,Z 285.51,A -85,B 0,C 180,E1 -23369.148,E2 -23369.148} C_VEL
LIN {X 0,Y 164.384,Z 285.5,A -85,B 0,C 180,E1 -23374.706,E2 -23374.706} C_VEL
LIN {X 0,Y 164.4,Z 285.497,A -85,B 0,C 180,E1 -23380.13,E2 -23380.13} C_VEL
LIN {X 0,Y 164.472,Z 285.489,A -85,B 0,C 180,E1 -23385.16,E2 -23385.16} C_VEL
LIN {X 0,Y 164.755,Z 285.454,A -85,B 0,C 180,E1 -23390.191,E2 -23390.191} C_VEL
LIN {X 0,Y 164.815,Z 285.456,A -85,B 0,C 180,E1 -23392.665,E2 -23392.665} C_VEL
LIN {X 0,Y 165.27,Z 285.373,A -85,B 0,C 180,E1 -23400.014,E2 -23400.014} C_VEL
LIN {X 0,Y 164.821,Z 285.455,A -85,B 0,C 180,E1 -23407.363,E2 -23407.363} C_VEL
LIN {X 0,Y 164.706,Z 285.469,A -85,B 0,C 180,E1 -23411.07,E2 -23411.07} C_VEL
LIN {X 0,Y 164.435,Z 285.503,A -85,B 0,C 180,E1 -23417.422,E2 -23417.422} C_VEL
LIN {X 0,Y 164.43,Z 285.505,A -85,B 0,C 180,E1 -23420.009,E2 -23420.009} C_VEL
LIN {X 0,Y 164.581,Z 287.095,A -85,B 0,C 180,E1 -23426.268,E2 -23426.268} C_VEL
LIN {X 0,Y 164.759,Z 288.724,A -85,B 0,C 180,E1 -23431.449,E2 -23431.449} C_VEL
LIN {X 0,Y 165.007,Z 290.52,A -85,B 0,C 180,E1 -23436.62,E2 -23436.62} C_VEL
LIN {X 0,Y 165.253,Z 292.516,A -85,B 0,C 180,E1 -23441.572,E2 -23441.572} C_VEL
LIN {X 0,Y 166.301,Z 295.654,A -85,B 0,C 180,E1 -23442.268,E2 -23442.268} C_VEL
LIN {X 0,Y 168.187,Z 298.493,A -85,B 0,C 180,E1 -23443.268,E2 -23443.268} C_VEL
LIN {X 0,Y 170.012,Z 302.377,A -85,B 0,C 180,E1 -23444.377,E2 -23444.377} C_VEL
LIN {X 0,Y 172.94,Z 309.753,A -85,B 0,C 180,E1 -23446.303,E2 -23446.303} C_VEL
LIN {X 0,Y 175.527,Z 319.024,A -85,B 0,C 180,E1 -23448.548,E2 -23448.548} C_VEL
LIN {X 0,Y 177.404,Z 329.158,A -85,B 0,C 180,E1 -23451.01,E2 -23451.01} C_VEL
LIN {X 0,Y 178.3,Z 338.21,A -85,B 0,C 180,E1 -23453.286,E2 -23453.286} C_VEL
LIN {X 0,Y 178.428,Z 347.623,A -85,B 0,C 180,E1 -23455.826,E2 -23455.826} C_VEL
LIN {X 0,Y 178.076,Z 354.406,A -85,B 0,C 180,E1 -23457.806,E2 -23457.806} C_VEL
LIN {X 0,Y 177.581,Z 358.278,A -85,B 0,C 180,E1 -23459.037,E2 -23459.037} C_VEL
LIN {X 0,Y 175.008,Z 365.21,A -85,B 0,C 180,E1 -23461.191,E2 -23461.191} C_VEL
LIN {X 0,Y 172.105,Z 372.257,A -85,B 0,C 180,E1 -23463.828,E2 -23463.828} C_VEL
LIN {X 0,Y 169.419,Z 378.643,A -85,B 0,C 180,E1 -23466.791,E2 -23466.791} C_VEL
LIN {X 0,Y 166.702,Z 384.668,A -85,B 0,C 180,E1 -23470.29,E2 -23470.29} C_VEL
LIN {X 0,Y 164.531,Z 389.415,A -85,B 0,C 180,E1 -23473.88,E2 -23473.88} C_VEL
LIN {X 0,Y 163.142,Z 393.033,A -85,B 0,C 180,E1 -23477.562,E2 -23477.562} C_VEL
LIN {X 0,Y 162.466,Z 394.837,A -85,B 0,C 180,E1 -23480.036,E2 -23480.036} C_VEL
LIN {X 0,Y 161.88,Z 397.299,A -85,B 0,C 180,E1 -23485.019,E2 -23485.019} C_VEL
LIN {X 0,Y 161.792,Z 397.966,A -85,B 0,C 180,E1 -23487.818,E2 -23487.818} C_VEL
LIN {X 0,Y 161.876,Z 398.052,A -85,B 0,C 180,E1 -23490,E2 -23490} C_VEL
LIN {X 0,Y 161.791,Z 397.893,A -85,B 0,C 180,E1 -23492.49,E2 -23492.49} C_VEL
LIN {X 0,Y 161.88,Z 397.299,A -85,B 0,C 180,E1 -23494.981,E2 -23494.981} C_VEL
LIN {X 0,Y 162.469,Z 394.838,A -85,B 0,C 180,E1 -23499.964,E2 -23499.964} C_VEL
LIN {X 0,Y 163.534,Z 391.879,A -85,B 0,C 180,E1 -23503.672,E2 -23503.672} C_VEL
LIN {X 0,Y 165.154,Z 387.882,A -85,B 0,C 180,E1 -23507.33,E2 -23507.33} C_VEL
LIN {X 0,Y 167.551,Z 382.751,A -85,B 0,C 180,E1 -23510.887,E2 -23510.887} C_VEL
LIN {X 0,Y 169.954,Z 377.488,A -85,B 0,C 180,E1 -23513.777,E2 -23513.777} C_VEL
LIN {X 0,Y 171.805,Z 373.097,A -85,B 0,C 180,E1 -23515.825,E2 -23515.825} C_VEL
LIN {X 0,Y 174.352,Z 366.837,A -85,B 0,C 180,E1 -23518.27,E2 -23518.27} C_VEL
LIN {X 0,Y 177.019,Z 360.203,A -85,B 0,C 180,E1 -23520.41,E2 -23520.41} C_VEL
LIN {X 0,Y 177.785,Z 356.341,A -85,B 0,C 180,E1 -23521.586,E2 -23521.586} C_VEL
LIN {X 0,Y 178.337,Z 349.788,A -85,B 0,C 180,E1 -23523.553,E2 -23523.553} C_VEL
LIN {X 0,Y 178.417,Z 342.703,A -85,B 0,C 180,E1 -23525.54,E2 -23525.54} C_VEL
LIN {X 0,Y 177.931,Z 333.992,A -85,B 0,C 180,E1 -23527.801,E2 -23527.801} C_VEL
LIN {X 0,Y 177.007,Z 326.259,A -85,B 0,C 180,E1 -23529.71,E2 -23529.71} C_VEL
LIN {X 0,Y 175.589,Z 321.864,A -85,B 0,C 180,E1 -23530.906,E2 -23530.906} C_VEL
LIN {X 0,Y 173.414,Z 318.089,A -85,B 0,C 180,E1 -23532.236,E2 -23532.236} C_VEL
LIN {X 0,Y 166.401,Z 308.852,A -85,B 0,C 180,E1 -23536.004,E2 -23536.004} C_VEL
LIN {X 0,Y 164.969,Z 306.187,A -85,B 0,C 180,E1 -23536.924,E2 -23536.924} C_VEL
LIN {X 0,Y 163.17,Z 302.34,A -85,B 0,C 180,E1 -23538.101,E2 -23538.101} C_VEL
LIN {X 0,Y 161.347,Z 298.631,A -85,B 0,C 180,E1 -23539.318,E2 -23539.318} C_VEL
LIN {X 0,Y 160.673,Z 297.376,A -85,B 0,C 180,E1 -23539.766,E2 -23539.766} C_VEL
LIN {X 0,Y 158.65,Z 294.32,A -85,B 0,C 180,E1 -23540.961,E2 -23540.961} C_VEL
LIN {X 0,Y 158.024,Z 292.121,A -85,B 0,C 180,E1 -23541.475,E2 -23541.475} C_VEL
LIN {X 0,Y 157.876,Z 291.003,A -85,B 0,C 180,E1 -23544.625,E2 -23544.625} C_VEL
LIN {X 0,Y 157.749,Z 289.955,A -85,B 0,C 180,E1 -23547.829,E2 -23547.829} C_VEL
LIN {X 0,Y 157.556,Z 288.256,A -85,B 0,C 180,E1 -23553.494,E2 -23553.494} C_VEL
LIN {X 0,Y 157.402,Z 286.665,A -85,B 0,C 180,E1 -23559.658,E2 -23559.658} C_VEL
LIN {X 0,Y 157.412,Z 286.378,A -85,B 0,C 180,E1 -23564.447,E2 -23564.447} C_VEL
LIN {X 0,Y 157.69,Z 286.343,A -85,B 0,C 180,E1 -23569.716,E2 -23569.716} C_VEL
LIN {X 0,Y 157.76,Z 286.334,A -85,B 0,C 180,E1 -23572.305,E2 -23572.305} C_VEL
LIN {X 0,Y 158.232,Z 286.248,A -85,B 0,C 180,E1 -23579.985,E2 -23579.985} C_VEL
LIN {X 0,Y 157.753,Z 286.334,A -85,B 0,C 180,E1 -23587.665,E2 -23587.665} C_VEL
LIN {X 0,Y 157.621,Z 286.347,A -85,B 0,C 180,E1 -23591.212,E2 -23591.212} C_VEL
LIN {X 0,Y 157.404,Z 286.37,A -85,B 0,C 180,E1 -23595.523,E2 -23595.523} C_VEL
LIN {X 0,Y 157.295,Z 286.384,A -85,B 0,C 180,E1 -23600.926,E2 -23600.926} C_VEL
LIN {X 0,Y 157.287,Z 286.39,A -85,B 0,C 180,E1 -23606.666,E2 -23606.666} C_VEL
LIN {X 0,Y 157.251,Z 286.398,A -85,B 0,C 180,E1 -23612.413,E2 -23612.413} C_VEL
LIN {X 0,Y 157.262,Z 286.396,A -85,B 0,C 180,E1 -23617.461,E2 -23617.461} C_VEL
LIN {X 0,Y 157.239,Z 286.397,A -85,B 0,C 180,E1 -23618.167,E2 -23618.167} C_VEL
LIN {X 0,Y 158.243,Z 289.229,A -85,B 0,C 180,E1 -23618.937,E2 -23618.937} C_VEL
LIN {X 0,Y 160.649,Z 291.884,A -85,B 0,C 180,E1 -23620.319,E2 -23620.319} C_VEL
LIN {X 0,Y 162.405,Z 295.013,A -85,B 0,C 180,E1 -23621.479,E2 -23621.479} C_VEL
LIN {X 0,Y 163.792,Z 296.924,A -85,B 0,C 180,E1 -23622.286,E2 -23622.286} C_VEL
LIN {X 0,Y 167.602,Z 303.396,A -85,B 0,C 180,E1 -23624.678,E2 -23624.678} C_VEL
LIN {X 0,Y 171.717,Z 311.407,A -85,B 0,C 180,E1 -23627.427,E2 -23627.427} C_VEL
LIN {X 0,Y 175.806,Z 321.462,A -85,B 0,C 180,E1 -23630.691,E2 -23630.691} C_VEL
LIN {X 0,Y 178.379,Z 329.814,A -85,B 0,C 180,E1 -23633.335,E2 -23633.335} C_VEL
LIN {X 0,Y 180.181,Z 337.022,A -85,B 0,C 180,E1 -23635.673,E2 -23635.673} C_VEL
LIN {X 0,Y 182.243,Z 346.837,A -85,B 0,C 180,E1 -23639.157,E2 -23639.157} C_VEL
LIN {X 0,Y 184.672,Z 354.026,A -85,B 0,C 180,E1 -23642.157,E2 -23642.157} C_VEL
LIN {X 0,Y 187.796,Z 359.948,A -85,B 0,C 180,E1 -23645.015,E2 -23645.015} C_VEL
LIN {X 0,Y 192.646,Z 366.388,A -85,B 0,C 180,E1 -23648.604,E2 -23648.604} C_VEL
LIN {X 0,Y 197.106,Z 370.643,A -85,B 0,C 180,E1 -23651.283,E2 -23651.283} C_VEL
LIN {X 0,Y 203.904,Z 375.418,A -85,B 0,C 180,E1 -23654.758,E2 -23654.758} C_VEL
LIN {X 0,Y 212.664,Z 379.769,A -85,B 0,C 180,E1 -23658.564,E2 -23658.564} C_VEL
LIN {X 0,Y 220.249,Z 382.475,A -85,B 0,C 180,E1 -23661.471,E2 -23661.471} C_VEL
LIN {X 0,Y 226.22,Z 384.124,A -85,B 0,C 180,E1 -23663.672,E2 -23663.672} C_VEL
LIN {X 0,Y 233.732,Z 385.578,A -85,B 0,C 180,E1 -23666.552,E2 -23666.552} C_VEL
LIN {X 0,Y 237.098,Z 386.049,A -85,B 0,C 180,E1 -23668.301,E2 -23668.301} C_VEL
LIN {X 0,Y 238.913,Z 386.157,A -85,B 0,C 180,E1 -23669.331,E2 -23669.331} C_VEL
LIN {X 0,Y 239.783,Z 386.146,A -85,B 0,C 180,E1 -23670,E2 -23670} C_VEL
LIN {X 0,Y 238.913,Z 386.157,A -85,B 0,C 180,E1 -23670.667,E2 -23670.667} C_VEL
LIN {X 0,Y 237.092,Z 386.049,A -85,B 0,C 180,E1 -23671.699,E2 -23671.699} C_VEL
LIN {X 0,Y 233.732,Z 385.578,A -85,B 0,C 180,E1 -23673.448,E2 -23673.448} C_VEL
LIN {X 0,Y 226.224,Z 384.116,A -85,B 0,C 180,E1 -23676.339,E2 -23676.339} C_VEL
LIN {X 0,Y 218.312,Z 381.877,A -85,B 0,C 180,E1 -23679.263,E2 -23679.263} C_VEL
LIN {X 0,Y 209.063,Z 378.197,A -85,B 0,C 180,E1 -23682.934,E2 -23682.934} C_VEL
LIN {X 0,Y 200.508,Z 373.2,A -85,B 0,C 180,E1 -23686.893,E2 -23686.893} C_VEL
LIN {X 0,Y 194.609,Z 368.373,A -85,B 0,C 180,E1 -23690.169,E2 -23690.169} C_VEL
LIN {X 0,Y 190.563,Z 364.008,A -85,B 0,C 180,E1 -23692.819,E2 -23692.819} C_VEL
LIN {X 0,Y 185.911,Z 356.515,A -85,B 0,C 180,E1 -23696.676,E2 -23696.676} C_VEL
LIN {X 0,Y 183.528,Z 350.737,A -85,B 0,C 180,E1 -23699.279,E2 -23699.279} C_VEL
LIN {X 0,Y 181.305,Z 342.861,A -85,B 0,C 180,E1 -23702.334,E2 -23702.334} C_VEL
LIN {X 0,Y 179.55,Z 334.21,A -85,B 0,C 180,E1 -23705.233,E2 -23705.233} C_VEL
LIN {X 0,Y 177.169,Z 325.663,A -85,B 0,C 180,E1 -23707.989,E2 -23707.989} C_VEL
LIN {X 0,Y 174.031,Z 316.832,A -85,B 0,C 180,E1 -23710.807,E2 -23710.807} C_VEL
LIN {X 0,Y 170.068,Z 308.122,A -85,B 0,C 180,E1 -23713.706,E2 -23713.706} C_VEL
LIN {X 0,Y 166.051,Z 300.554,A -85,B 0,C 180,E1 -23716.363,E2 -23716.363} C_VEL
LIN {X 0,Y 163.466,Z 296.321,A -85,B 0,C 180,E1 -23717.922,E2 -23717.922} C_VEL
LIN {X 0,Y 160.999,Z 292.734,A -85,B 0,C 180,E1 -23719.414,E2 -23719.414} C_VEL
LIN {X 0,Y 160.152,Z 291.23,A -85,B 0,C 180,E1 -23719.986,E2 -23719.986} C_VEL
LIN {X 0,Y 158.144,Z 289.03,A -85,B 0,C 180,E1 -23721.137,E2 -23721.137} C_VEL
LIN {X 0,Y 157.291,Z 286.721,A -85,B 0,C 180,E1 -23721.77,E2 -23721.77} C_VEL
LIN {X 0,Y 157.256,Z 286.395,A -85,B 0,C 180,E1 -23721.916,E2 -23721.916} C_VEL
LIN {X 0,Y 157.263,Z 286.394,A -85,B 0,C 180,E1 -23724.503,E2 -23724.503} C_VEL
LIN {X 0,Y 157.268,Z 286.395,A -85,B 0,C 180,E1 -23728.109,E2 -23728.109} C_VEL
LIN {X 0,Y 157.293,Z 286.389,A -85,B 0,C 180,E1 -23733.479,E2 -23733.479} C_VEL
LIN {X 0,Y 157.343,Z 286.376,A -85,B 0,C 180,E1 -23739.716,E2 -23739.716} C_VEL
LIN {X 0,Y 157.404,Z 286.37,A -85,B 0,C 180,E1 -23744.477,E2 -23744.477} C_VEL
LIN {X 0,Y 157.677,Z 286.336,A -85,B 0,C 180,E1 -23749.746,E2 -23749.746} C_VEL
LIN {X 0,Y 157.753,Z 286.334,A -85,B 0,C 180,E1 -23752.335,E2 -23752.335} C_VEL
LIN {X 0,Y 158.232,Z 286.248,A -85,B 0,C 180,E1 -23760.015,E2 -23760.015} C_VEL
LIN {X 0,Y 157.76,Z 286.335,A -85,B 0,C 180,E1 -23767.695,E2 -23767.695} C_VEL
LIN {X 0,Y 157.635,Z 286.351,A -85,B 0,C 180,E1 -23771.237,E2 -23771.237} C_VEL
LIN {X 0,Y 157.412,Z 286.379,A -85,B 0,C 180,E1 -23775.553,E2 -23775.553} C_VEL
LIN {X 0,Y 157.402,Z 286.661,A -85,B 0,C 180,E1 -23780.343,E2 -23780.343} C_VEL
LIN {X 0,Y 157.556,Z 288.254,A -85,B 0,C 180,E1 -23786.506,E2 -23786.506} C_VEL
LIN {X 0,Y 157.753,Z 290.006,A -85,B 0,C 180,E1 -23792.333,E2 -23792.333} C_VEL
LIN {X 0,Y 157.969,Z 291.524,A -85,B 0,C 180,E1 -23796.794,E2 -23796.794} C_VEL
LIN {X 0,Y 158.066,Z 292.327,A -85,B 0,C 180,E1 -23798.583,E2 -23798.583} C_VEL
LIN {X 0,Y 159.102,Z 295.261,A -85,B 0,C 180,E1 -23799.325,E2 -23799.325} C_VEL
LIN {X 0,Y 161.227,Z 298.301,A -85,B 0,C 180,E1 -23800.588,E2 -23800.588} C_VEL
LIN {X 0,Y 162.938,Z 302.002,A -85,B 0,C 180,E1 -23801.765,E2 -23801.765} C_VEL
LIN {X 0,Y 163.94,Z 303.786,A -85,B 0,C 180,E1 -23802.381,E2 -23802.381} C_VEL
LIN {X 0,Y 166.739,Z 310.522,A -85,B 0,C 180,E1 -23804.402,E2 -23804.402} C_VEL
LIN {X 0,Y 169.165,Z 318.501,A -85,B 0,C 180,E1 -23806.562,E2 -23806.562} C_VEL
LIN {X 0,Y 170.987,Z 327.943,A -85,B 0,C 180,E1 -23809.019,E2 -23809.019} C_VEL
LIN {X 0,Y 171.991,Z 337.974,A -85,B 0,C 180,E1 -23811.702,E2 -23811.702} C_VEL
LIN {X 0,Y 172.136,Z 347.502,A -85,B 0,C 180,E1 -23814.425,E2 -23814.425} C_VEL
LIN {X 0,Y 171.525,Z 356.121,A -85,B 0,C 180,E1 -23817.119,E2 -23817.119} C_VEL
LIN {X 0,Y 170.873,Z 359.989,A -85,B 0,C 180,E1 -23818.372,E2 -23818.372} C_VEL
LIN {X 0,Y 166.858,Z 369.576,A -85,B 0,C 180,E1 -23821.716,E2 -23821.716} C_VEL
LIN {X 0,Y 163.992,Z 376.119,A -85,B 0,C 180,E1 -23824.624,E2 -23824.624} C_VEL
LIN {X 0,Y 161.819,Z 380.621,A -85,B 0,C 180,E1 -23826.991,E2 -23826.991} C_VEL
LIN {X 0,Y 159.186,Z 386.117,A -85,B 0,C 180,E1 -23830.663,E2 -23830.663} C_VEL
LIN {X 0,Y 157.101,Z 390.446,A -85,B 0,C 180,E1 -23834.43,E2 -23834.43} C_VEL
LIN {X 0,Y 156.169,Z 392.82,A -85,B 0,C 180,E1 -23836.997,E2 -23836.997} C_VEL
LIN {X 0,Y 155.465,Z 394.626,A -85,B 0,C 180,E1 -23839.582,E2 -23839.582} C_VEL
LIN {X 0,Y 154.784,Z 397.087,A -85,B 0,C 180,E1 -23844.79,E2 -23844.79} C_VEL
LIN {X 0,Y 154.715,Z 397.834,A -85,B 0,C 180,E1 -23848.305,E2 -23848.305} C_VEL
LIN {X 0,Y 154.697,Z 397.682,A -85,B 0,C 180,E1 -23852.604,E2 -23852.604} C_VEL
LIN {X 0,Y 154.786,Z 397.087,A -85,B 0,C 180,E1 -23855.21,E2 -23855.21} C_VEL
LIN {X 0,Y 155.467,Z 394.626,A -85,B 0,C 180,E1 -23860.417,E2 -23860.417} C_VEL
LIN {X 0,Y 156.608,Z 391.667,A -85,B 0,C 180,E1 -23864.289,E2 -23864.289} C_VEL
LIN {X 0,Y 158.376,Z 387.671,A -85,B 0,C 180,E1 -23868.097,E2 -23868.097} C_VEL
LIN {X 0,Y 160.897,Z 382.539,A -85,B 0,C 180,E1 -23871.794,E2 -23871.794} C_VEL
LIN {X 0,Y 163.444,Z 377.275,A -85,B 0,C 180,E1 -23874.786,E2 -23874.786} C_VEL
LIN {X 0,Y 166.207,Z 370.952,A -85,B 0,C 180,E1 -23877.718,E2 -23877.718} C_VEL
LIN {X 0,Y 168.785,Z 364.998,A -85,B 0,C 180,E1 -23879.977,E2 -23879.977} C_VEL
LIN {X 0,Y 170.83,Z 359.988,A -85,B 0,C 180,E1 -23881.637,E2 -23881.637} C_VEL
LIN {X 0,Y 171.898,Z 352.087,A -85,B 0,C 180,E1 -23884.205,E2 -23884.205} C_VEL
LIN {X 0,Y 172.162,Z 342.548,A -85,B 0,C 180,E1 -23887.021,E2 -23887.021} C_VEL
LIN {X 0,Y 171.686,Z 333.949,A -85,B 0,C 180,E1 -23889.391,E2 -23889.391} C_VEL
LIN {X 0,Y 170.648,Z 325.666,A -85,B 0,C 180,E1 -23891.576,E2 -23891.576} C_VEL
LIN {X 0,Y 168.275,Z 315.041,A -85,B 0,C 180,E1 -23894.345,E2 -23894.345} C_VEL
LIN {X 0,Y 164.969,Z 306.187,A -85,B 0,C 180,E1 -23896.924,E2 -23896.924} C_VEL
LIN {X 0,Y 163.397,Z 303.778,A -85,B 0,C 180,E1 -23897.869,E2 -23897.869} C_VEL
LIN {X 0,Y 159.933,Z 301.022,A -85,B 0,C 180,E1 -23899.62,E2 -23899.62} C_VEL
LIN {X 0,Y 154.004,Z 297.578,A -85,B 0,C 180,E1 -23902.716,E2 -23902.716} C_VEL
LIN {X 0,Y 151.766,Z 294.744,A -85,B 0,C 180,E1 -23904.206,E2 -23904.206} C_VEL
LIN {X 0,Y 150.796,Z 291.738,A -85,B 0,C 180,E1 -23905.169,E2 -23905.169} C_VEL
LIN {X 0,Y 150.608,Z 290.551,A -85,B 0,C 180,E1 -23909.1,E2 -23909.1} C_VEL
LIN {X 0,Y 150.514,Z 289.581,A -85,B 0,C 180,E1 -23912.518,E2 -23912.518} C_VEL
LIN {X 0,Y 150.38,Z 288.177,A -85,B 0,C 180,E1 -23918.03,E2 -23918.03} C_VEL
LIN {X 0,Y 150.339,Z 287.53,A -85,B 0,C 180,E1 -23920.884,E2 -23920.884} C_VEL
LIN {X 0,Y 150.409,Z 287.25,A -85,B 0,C 180,E1 -23926.474,E2 -23926.474} C_VEL
LIN {X 0,Y 150.61,Z 287.225,A -85,B 0,C 180,E1 -23929.227,E2 -23929.227} C_VEL
LIN {X 0,Y 150.699,Z 287.215,A -85,B 0,C 180,E1 -23931.942,E2 -23931.942} C_VEL
LIN {X 0,Y 151.193,Z 287.122,A -85,B 0,C 180,E1 -23939.985,E2 -23939.985} C_VEL
LIN {X 0,Y 150.691,Z 287.213,A -85,B 0,C 180,E1 -23948.027,E2 -23948.027} C_VEL
LIN {X 0,Y 150.563,Z 287.227,A -85,B 0,C 180,E1 -23951.415,E2 -23951.415} C_VEL
LIN {X 0,Y 150.308,Z 287.257,A -85,B 0,C 180,E1 -23956.275,E2 -23956.275} C_VEL
LIN {X 0,Y 150.267,Z 287.258,A -85,B 0,C 180,E1 -23960.71,E2 -23960.71} C_VEL
LIN {X 0,Y 150.219,Z 287.274,A -85,B 0,C 180,E1 -23967.265,E2 -23967.265} C_VEL
LIN {X 0,Y 150.191,Z 287.277,A -85,B 0,C 180,E1 -23972.619,E2 -23972.619} C_VEL
LIN {X 0,Y 150.181,Z 287.332,A -85,B 0,C 180,E1 -23974.701,E2 -23974.701} C_VEL
LIN {X 0,Y 151.139,Z 289.987,A -85,B 0,C 180,E1 -23975.517,E2 -23975.517} C_VEL
LIN {X 0,Y 153.126,Z 292.137,A -85,B 0,C 180,E1 -23976.862,E2 -23976.862} C_VEL
LIN {X 0,Y 153.771,Z 292.945,A -85,B 0,C 180,E1 -23977.312,E2 -23977.312} C_VEL
LIN {X 0,Y 155.538,Z 296.079,A -85,B 0,C 180,E1 -23978.643,E2 -23978.643} C_VEL
LIN {X 0,Y 156.927,Z 297.776,A -85,B 0,C 180,E1 -23979.53,E2 -23979.53} C_VEL
LIN {X 0,Y 161.869,Z 306.138,A -85,B 0,C 180,E1 -23983.036,E2 -23983.036} C_VEL
LIN {X 0,Y 165.86,Z 314.082,A -85,B 0,C 180,E1 -23986.059,E2 -23986.059} C_VEL
LIN {X 0,Y 168.722,Z 321.149,A -85,B 0,C 180,E1 -23988.546,E2 -23988.546} C_VEL
LIN {X 0,Y 171.542,Z 329.626,A -85,B 0,C 180,E1 -23991.49,E2 -23991.49} C_VEL
LIN {X 0,Y 173.686,Z 338.318,A -85,B 0,C 180,E1 -23994.536,E2 -23994.536} C_VEL
LIN {X 0,Y 175.281,Z 347.268,A -85,B 0,C 180,E1 -23997.857,E2 -23997.857} C_VEL
LIN {X 0,Y 177.126,Z 354.045,A -85,B 0,C 180,E1 -24000.766,E2 -24000.766} C_VEL
LIN {X 0,Y 179.905,Z 360.388,A -85,B 0,C 180,E1 -24003.924,E2 -24003.924} C_VEL
LIN {X 0,Y 184.164,Z 366.654,A -85,B 0,C 180,E1 -24007.567,E2 -24007.567} C_VEL
LIN {X 0,Y 189.523,Z 372.007,A -85,B 0,C 180,E1 -24011.18,E2 -24011.18} C_VEL
LIN {X 0,Y 196.446,Z 376.757,A -85,B 0,C 180,E1 -24014.945,E2 -24014.945} C_VEL
LIN {X 0,Y 203.149,Z 380.053,A -85,B 0,C 180,E1 -24018.02,E2 -24018.02} C_VEL
LIN {X 0,Y 212.904,Z 383.367,A -85,B 0,C 180,E1 -24021.911,E2 -24021.911} C_VEL
LIN {X 0,Y 219.873,Z 384.966,A -85,B 0,C 180,E1 -24024.497,E2 -24024.497} C_VEL
LIN {X 0,Y 225.258,Z 385.868,A -85,B 0,C 180,E1 -24026.512,E2 -24026.512} C_VEL
LIN {X 0,Y 229.115,Z 386.286,A -85,B 0,C 180,E1 -24028.242,E2 -24028.242} C_VEL
LIN {X 0,Y 232.348,Z 386.363,A -85,B 0,C 180,E1 -24030,E2 -24030} C_VEL
LIN {X 0,Y 229.111,Z 386.286,A -85,B 0,C 180,E1 -24031.758,E2 -24031.758} C_VEL
LIN {X 0,Y 225.045,Z 385.837,A -85,B 0,C 180,E1 -24033.581,E2 -24033.581} C_VEL
LIN {X 0,Y 218.956,Z 384.788,A -85,B 0,C 180,E1 -24035.855,E2 -24035.855} C_VEL
LIN {X 0,Y 212.909,Z 383.358,A -85,B 0,C 180,E1 -24038.097,E2 -24038.097} C_VEL
LIN {X 0,Y 203.155,Z 380.053,A -85,B 0,C 180,E1 -24041.979,E2 -24041.979} C_VEL
LIN {X 0,Y 194.256,Z 375.478,A -85,B 0,C 180,E1 -24046.184,E2 -24046.184} C_VEL
LIN {X 0,Y 186.236,Z 369.016,A -85,B 0,C 180,E1 -24050.921,E2 -24050.921} C_VEL
LIN {X 0,Y 181.495,Z 362.99,A -85,B 0,C 180,E1 -24054.622,E2 -24054.622} C_VEL
LIN {X 0,Y 178.552,Z 357.483,A -85,B 0,C 180,E1 -24057.578,E2 -24057.578} C_VEL
LIN {X 0,Y 176.247,Z 350.989,A -85,B 0,C 180,E1 -24060.612,E2 -24060.612} C_VEL
LIN {X 0,Y 174.544,Z 343.238,A -85,B 0,C 180,E1 -24063.707,E2 -24063.707} C_VEL
LIN {X 0,Y 172.768,Z 334.402,A -85,B 0,C 180,E1 -24066.853,E2 -24066.853} C_VEL
LIN {X 0,Y 170.196,Z 325.295,A -85,B 0,C 180,E1 -24069.999,E2 -24069.999} C_VEL
LIN {X 0,Y 166.597,Z 315.806,A -85,B 0,C 180,E1 -24073.329,E2 -24073.329} C_VEL
LIN {X 0,Y 162.756,Z 307.851,A -85,B 0,C 180,E1 -24076.322,E2 -24076.322} C_VEL
LIN {X 0,Y 158.178,Z 299.964,A -85,B 0,C 180,E1 -24079.6,E2 -24079.6} C_VEL
LIN {X 0,Y 156.282,Z 296.844,A -85,B 0,C 180,E1 -24080.899,E2 -24080.899} C_VEL
LIN {X 0,Y 154.053,Z 293.722,A -85,B 0,C 180,E1 -24082.428,E2 -24082.428} C_VEL
LIN {X 0,Y 153.407,Z 292.341,A -85,B 0,C 180,E1 -24082.964,E2 -24082.964} C_VEL
LIN {X 0,Y 151.244,Z 290.14,A -85,B 0,C 180,E1 -24084.409,E2 -24084.409} C_VEL
LIN {X 0,Y 150.232,Z 287.647,A -85,B 0,C 180,E1 -24085.261,E2 -24085.261} C_VEL
LIN {X 0,Y 150.176,Z 287.279,A -85,B 0,C 180,E1 -24085.45,E2 -24085.45} C_VEL
LIN {X 0,Y 150.182,Z 287.276,A -85,B 0,C 180,E1 -24089.039,E2 -24089.039} C_VEL
LIN {X 0,Y 150.219,Z 287.274,A -85,B 0,C 180,E1 -24092.735,E2 -24092.735} C_VEL
LIN {X 0,Y 150.267,Z 287.258,A -85,B 0,C 180,E1 -24099.29,E2 -24099.29} C_VEL
LIN {X 0,Y 150.308,Z 287.257,A -85,B 0,C 180,E1 -24103.725,E2 -24103.725} C_VEL
LIN {X 0,Y 150.597,Z 287.219,A -85,B 0,C 180,E1 -24109.258,E2 -24109.258} C_VEL
LIN {X 0,Y 150.691,Z 287.213,A -85,B 0,C 180,E1 -24111.973,E2 -24111.973} C_VEL
LIN {X 0,Y 151.193,Z 287.122,A -85,B 0,C 180,E1 -24120.015,E2 -24120.015} C_VEL
LIN {X 0,Y 150.683,Z 287.217,A -85,B 0,C 180,E1 -24128.059,E2 -24128.059} C_VEL
LIN {X 0,Y 150.578,Z 287.23,A -85,B 0,C 180,E1 -24131.442,E2 -24131.442} C_VEL
LIN {X 0,Y 150.318,Z 287.261,A -85,B 0,C 180,E1 -24136.307,E2 -24136.307} C_VEL
LIN {X 0,Y 150.384,Z 287.905,A -85,B 0,C 180,E1 -24140.827,E2 -24140.827} C_VEL
LIN {X 0,Y 150.45,Z 288.891,A -85,B 0,C 180,E1 -24144.876,E2 -24144.876} C_VEL
LIN {X 0,Y 150.521,Z 289.682,A -85,B 0,C 180,E1 -24147.85,E2 -24147.85} C_VEL
LIN {X 0,Y 150.732,Z 291.197,A -85,B 0,C 180,E1 -24152.939,E2 -24152.939} C_VEL
LIN {X 0,Y 150.855,Z 292.081,A -85,B 0,C 180,E1 -24155.019,E2 -24155.019} C_VEL
LIN {X 0,Y 151.977,Z 295.101,A -85,B 0,C 180,E1 -24155.941,E2 -24155.941} C_VEL
LIN {X 0,Y 154.322,Z 298.193,A -85,B 0,C 180,E1 -24157.53,E2 -24157.53} C_VEL
LIN {X 0,Y 156.052,Z 301.89,A -85,B 0,C 180,E1 -24158.879,E2 -24158.879} C_VEL
LIN {X 0,Y 157.145,Z 303.596,A -85,B 0,C 180,E1 -24159.607,E2 -24159.607} C_VEL
LIN {X 0,Y 160.963,Z 312.206,A -85,B 0,C 180,E1 -24162.606,E2 -24162.606} C_VEL
LIN {X 0,Y 163.426,Z 320.373,A -85,B 0,C 180,E1 -24165.078,E2 -24165.078} C_VEL
LIN {X 0,Y 165.079,Z 329.742,A -85,B 0,C 180,E1 -24167.722,E2 -24167.722} C_VEL
LIN {X 0,Y 165.855,Z 338.239,A -85,B 0,C 180,E1 -24170.153,E2 -24170.153} C_VEL
LIN {X 0,Y 165.952,Z 346.117,A -85,B 0,C 180,E1 -24172.5,E2 -24172.5} C_VEL
LIN {X 0,Y 165.424,Z 354.381,A -85,B 0,C 180,E1 -24175.166,E2 -24175.166} C_VEL
LIN {X 0,Y 164.676,Z 359.771,A -85,B 0,C 180,E1 -24177.035,E2 -24177.035} C_VEL
LIN {X 0,Y 162.654,Z 364.786,A -85,B 0,C 180,E1 -24178.769,E2 -24178.769} C_VEL
LIN {X 0,Y 159.953,Z 370.74,A -85,B 0,C 180,E1 -24181.098,E2 -24181.098} C_VEL
LIN {X 0,Y 157.56,Z 375.906,A -85,B 0,C 180,E1 -24183.51,E2 -24183.51} C_VEL
LIN {X 0,Y 155.293,Z 380.409,A -85,B 0,C 180,E1 -24185.965,E2 -24185.965} C_VEL
LIN {X 0,Y 152.468,Z 385.905,A -85,B 0,C 180,E1 -24189.775,E2 -24189.775} C_VEL
LIN {X 0,Y 150.231,Z 390.233,A -85,B 0,C 180,E1 -24193.699,E2 -24193.699} C_VEL
LIN {X 0,Y 149.218,Z 392.607,A -85,B 0,C 180,E1 -24196.379,E2 -24196.379} C_VEL
LIN {X 0,Y 148.45,Z 394.413,A -85,B 0,C 180,E1 -24199.084,E2 -24199.084} C_VEL
LIN {X 0,Y 147.717,Z 396.876,A -85,B 0,C 180,E1 -24204.54,E2 -24204.54} C_VEL
LIN {X 0,Y 147.638,Z 397.628,A -85,B 0,C 180,E1 -24209.11,E2 -24209.11} C_VEL
LIN {X 0,Y 147.601,Z 397.47,A -85,B 0,C 180,E1 -24212.729,E2 -24212.729} C_VEL
LIN {X 0,Y 147.718,Z 396.876,A -85,B 0,C 180,E1 -24215.46,E2 -24215.46} C_VEL
LIN {X 0,Y 148.452,Z 394.413,A -85,B 0,C 180,E1 -24220.916,E2 -24220.916} C_VEL
LIN {X 0,Y 149.707,Z 391.454,A -85,B 0,C 180,E1 -24224.963,E2 -24224.963} C_VEL
LIN {X 0,Y 151.634,Z 387.459,A -85,B 0,C 180,E1 -24228.931,E2 -24228.931} C_VEL
LIN {X 0,Y 154.276,Z 382.326,A -85,B 0,C 180,E1 -24232.781,E2 -24232.781} C_VEL
LIN {X 0,Y 156.993,Z 377.063,A -85,B 0,C 180,E1 -24235.878,E2 -24235.878} C_VEL
LIN {X 0,Y 159.181,Z 372.361,A -85,B 0,C 180,E1 -24238.207,E2 -24238.207} C_VEL
LIN {X 0,Y 161.924,Z 366.413,A -85,B 0,C 180,E1 -24240.662,E2 -24240.662} C_VEL
LIN {X 0,Y 164.092,Z 361.53,A -85,B 0,C 180,E1 -24242.368,E2 -24242.368} C_VEL
LIN {X 0,Y 165.196,Z 356.108,A -85,B 0,C 180,E1 -24244.23,E2 -24244.23} C_VEL
LIN {X 0,Y 165.864,Z 348.416,A -85,B 0,C 180,E1 -24246.762,E2 -24246.762} C_VEL
LIN {X 0,Y 165.944,Z 340.751,A -85,B 0,C 180,E1 -24249.102,E2 -24249.102} C_VEL
LIN {X 0,Y 165.434,Z 332.442,A -85,B 0,C 180,E1 -24251.502,E2 -24251.502} C_VEL
LIN {X 0,Y 163.975,Z 323.001,A -85,B 0,C 180,E1 -24254.181,E2 -24254.181} C_VEL
LIN {X 0,Y 162.029,Z 315.231,A -85,B 0,C 180,E1 -24256.466,E2 -24256.466} C_VEL
LIN {X 0,Y 158.738,Z 307.019,A -85,B 0,C 180,E1 -24259.212,E2 -24259.212} C_VEL
LIN {X 0,Y 156.511,Z 302.517,A -85,B 0,C 180,E1 -24260.825,E2 -24260.825} C_VEL
LIN {X 0,Y 154.468,Z 298.693,A -85,B 0,C 180,E1 -24262.325,E2 -24262.325} C_VEL
LIN {X 0,Y 154.004,Z 297.578,A -85,B 0,C 180,E1 -24262.716,E2 -24262.716} C_VEL
LIN {X 0,Y 151.428,Z 295.577,A -85,B 0,C 180,E1 -24264.371,E2 -24264.371} C_VEL
LIN {X 0,Y 145.984,Z 292.336,A -85,B 0,C 180,E1 -24267.738,E2 -24267.738} C_VEL
LIN {X 0,Y 143.554,Z 291.417,A -85,B 0,C 180,E1 -24269.466,E2 -24269.466} C_VEL
LIN {X 0,Y 143.419,Z 290.282,A -85,B 0,C 180,E1 -24273.814,E2 -24273.814} C_VEL
LIN {X 0,Y 143.353,Z 288.863,A -85,B 0,C 180,E1 -24279.913,E2 -24279.913} C_VEL
LIN {X 0,Y 143.269,Z 288.274,A -85,B 0,C 180,E1 -24282.867,E2 -24282.867} C_VEL
LIN {X 0,Y 143.537,Z 288.106,A -85,B 0,C 180,E1 -24288.69,E2 -24288.69} C_VEL
LIN {X 0,Y 143.621,Z 288.095,A -85,B 0,C 180,E1 -24291.542,E2 -24291.542} C_VEL
LIN {X 0,Y 144.151,Z 287.997,A -85,B 0,C 180,E1 -24299.984,E2 -24299.984} C_VEL
LIN {X 0,Y 143.612,Z 288.091,A -85,B 0,C 180,E1 -24308.425,E2 -24308.425} C_VEL
LIN {X 0,Y 143.489,Z 288.109,A -85,B 0,C 180,E1 -24311.602,E2 -24311.602} C_VEL
LIN {X 0,Y 143.245,Z 288.142,A -85,B 0,C 180,E1 -24317.102,E2 -24317.102} C_VEL
LIN {X 0,Y 143.209,Z 288.139,A -85,B 0,C 180,E1 -24321.186,E2 -24321.186} C_VEL
LIN {X 0,Y 143.165,Z 288.152,A -85,B 0,C 180,E1 -24327.92,E2 -24327.92} C_VEL
LIN {X 0,Y 143.113,Z 288.158,A -85,B 0,C 180,E1 -24330.405,E2 -24330.405} C_VEL
LIN {X 0,Y 144.037,Z 290.84,A -85,B 0,C 180,E1 -24331.41,E2 -24331.41} C_VEL
LIN {X 0,Y 146.167,Z 293.121,A -85,B 0,C 180,E1 -24333.166,E2 -24333.166} C_VEL
LIN {X 0,Y 146.983,Z 293.996,A -85,B 0,C 180,E1 -24333.813,E2 -24333.813} C_VEL
LIN {X 0,Y 148.626,Z 296.986,A -85,B 0,C 180,E1 -24335.273,E2 -24335.273} C_VEL
LIN {X 0,Y 150.179,Z 298.733,A -85,B 0,C 180,E1 -24336.401,E2 -24336.401} C_VEL
LIN {X 0,Y 152.017,Z 301.904,A -85,B 0,C 180,E1 -24337.912,E2 -24337.912} C_VEL
LIN {X 0,Y 155.69,Z 308.06,A -85,B 0,C 180,E1 -24340.862,E2 -24340.862} C_VEL
LIN {X 0,Y 159.341,Z 315.329,A -85,B 0,C 180,E1 -24343.978,E2 -24343.978} C_VEL
LIN {X 0,Y 162.075,Z 321.82,A -85,B 0,C 180,E1 -24346.543,E2 -24346.543} C_VEL
LIN {X 0,Y 164.69,Z 329.493,A -85,B 0,C 180,E1 -24349.447,E2 -24349.447} C_VEL
LIN {X 0,Y 167.058,Z 338.965,A -85,B 0,C 180,E1 -24353.037,E2 -24353.037} C_VEL
LIN {X 0,Y 168.322,Z 346.822,A -85,B 0,C 180,E1 -24356.09,E2 -24356.09} C_VEL
LIN {X 0,Y 169.978,Z 354.666,A -85,B 0,C 180,E1 -24359.571,E2 -24359.571} C_VEL
LIN {X 0,Y 172.125,Z 360.652,A -85,B 0,C 180,E1 -24362.656,E2 -24362.656} C_VEL
LIN {X 0,Y 176.051,Z 367.174,A -85,B 0,C 180,E1 -24366.618,E2 -24366.618} C_VEL
LIN {X 0,Y 179.864,Z 371.533,A -85,B 0,C 180,E1 -24369.634,E2 -24369.634} C_VEL
LIN {X 0,Y 186.309,Z 376.49,A -85,B 0,C 180,E1 -24373.677,E2 -24373.677} C_VEL
LIN {X 0,Y 194.186,Z 380.552,A -85,B 0,C 180,E1 -24377.666,E2 -24377.666} C_VEL
LIN {X 0,Y 199.714,Z 382.641,A -85,B 0,C 180,E1 -24380.084,E2 -24380.084} C_VEL
LIN {X 0,Y 205.565,Z 384.259,A -85,B 0,C 180,E1 -24382.398,E2 -24382.398} C_VEL
LIN {X 0,Y 211.695,Z 385.451,A -85,B 0,C 180,E1 -24384.688,E2 -24384.688} C_VEL
LIN {X 0,Y 218.099,Z 386.288,A -85,B 0,C 180,E1 -24387.067,E2 -24387.067} C_VEL
LIN {X 0,Y 220.77,Z 386.533,A -85,B 0,C 180,E1 -24388.176,E2 -24388.176} C_VEL
LIN {X 0,Y 224.554,Z 386.591,A -85,B 0,C 180,E1 -24390,E2 -24390} C_VEL
LIN {X 0,Y 220.769,Z 386.533,A -85,B 0,C 180,E1 -24391.824,E2 -24391.824} C_VEL
LIN {X 0,Y 215.992,Z 386.107,A -85,B 0,C 180,E1 -24393.731,E2 -24393.731} C_VEL
LIN {X 0,Y 210.553,Z 385.24,A -85,B 0,C 180,E1 -24395.747,E2 -24395.747} C_VEL
LIN {X 0,Y 204.82,Z 384.065,A -85,B 0,C 180,E1 -24397.889,E2 -24397.889} C_VEL
LIN {X 0,Y 199.146,Z 382.456,A -85,B 0,C 180,E1 -24400.163,E2 -24400.163} C_VEL
LIN {X 0,Y 188.998,Z 378.083,A -85,B 0,C 180,E1 -24404.862,E2 -24404.862} C_VEL
LIN {X 0,Y 181.772,Z 373.2,A -85,B 0,C 180,E1 -24409.056,E2 -24409.056} C_VEL
LIN {X 0,Y 177.549,Z 369.12,A -85,B 0,C 180,E1 -24412.088,E2 -24412.088} C_VEL
LIN {X 0,Y 173.422,Z 363.023,A -85,B 0,C 180,E1 -24415.958,E2 -24415.958} C_VEL
LIN {X 0,Y 170.769,Z 357.037,A -85,B 0,C 180,E1 -24419.249,E2 -24419.249} C_VEL
LIN {X 0,Y 168.776,Z 349.523,A -85,B 0,C 180,E1 -24422.774,E2 -24422.774} C_VEL
LIN {X 0,Y 167.523,Z 341.558,A -85,B 0,C 180,E1 -24425.967,E2 -24425.967} C_VEL
LIN {X 0,Y 165.833,Z 333.937,A -85,B 0,C 180,E1 -24428.884,E2 -24428.884} C_VEL
LIN {X 0,Y 163.878,Z 326.959,A -85,B 0,C 180,E1 -24431.516,E2 -24431.516} C_VEL
LIN {X 0,Y 160.867,Z 318.643,A -85,B 0,C 180,E1 -24434.707,E2 -24434.707} C_VEL
LIN {X 0,Y 156.746,Z 309.987,A -85,B 0,C 180,E1 -24438.308,E2 -24438.308} C_VEL
LIN {X 0,Y 152.948,Z 303.19,A -85,B 0,C 180,E1 -24441.365,E2 -24441.365} C_VEL
LIN {X 0,Y 150.261,Z 298.963,A -85,B 0,C 180,E1 -24443.518,E2 -24443.518} C_VEL
LIN {X 0,Y 149.146,Z 297.525,A -85,B 0,C 180,E1 -24444.351,E2 -24444.351} C_VEL
LIN {X 0,Y 147.204,Z 294.587,A -85,B 0,C 180,E1 -24445.952,E2 -24445.952} C_VEL
LIN {X 0,Y 146.646,Z 293.426,A -85,B 0,C 180,E1 -24446.49,E2 -24446.49} C_VEL
LIN {X 0,Y 144.307,Z 291.247,A -85,B 0,C 180,E1 -24448.349,E2 -24448.349} C_VEL
LIN {X 0,Y 143.168,Z 288.532,A -85,B 0,C 180,E1 -24449.506,E2 -24449.506} C_VEL
LIN {X 0,Y 143.117,Z 288.158,A -85,B 0,C 180,E1 -24449.698,E2 -24449.698} C_VEL
LIN {X 0,Y 143.13,Z 288.149,A -85,B 0,C 180,E1 -24453.794,E2 -24453.794} C_VEL
LIN {X 0,Y 143.232,Z 288.133,A -85,B 0,C 180,E1 -24459.93,E2 -24459.93} C_VEL
LIN {X 0,Y 143.301,Z 288.127,A -85,B 0,C 180,E1 -24465.823,E2 -24465.823} C_VEL
LIN {X 0,Y 143.523,Z 288.103,A -85,B 0,C 180,E1 -24468.722,E2 -24468.722} C_VEL
LIN {X 0,Y 143.612,Z 288.091,A -85,B 0,C 180,E1 -24471.575,E2 -24471.575} C_VEL
LIN {X 0,Y 144.151,Z 287.997,A -85,B 0,C 180,E1 -24480.016,E2 -24480.016} C_VEL
